// TIA Portal V20 export
// export: Created 2025-12-01T14:57:38.3565208Z, ExportSetting None, DisplayName Totally Integrated Automation Portal, DisplayVersion V20 Update 3, DisplayName TIA Portal Openness, DisplayVersion V20 Update 3, DisplayName TIA Portal Version Control Interface, DisplayVersion V20 Update 3, DisplayName STEP 7 Professional, DisplayVersion V20 Update 3, DisplayName STEP 7 Safety, DisplayVersion V20 Update 2, DisplayName WinCC Basic/Comfort/Advanced, DisplayVersion V20 Update 3, DisplayName WinCC Professional, DisplayVersion V20 Update 3, DisplayName WinCC Unified, DisplayVersion V20 Update 3
FUNCTION_BLOCK "FB73_MesaBanda_DesPaletizadorCajasPlasticco"   // FB73, LAD
TITLE = Mesa de Banda DesPaletizador de Paletas
{ S7_Optimized_Access := 'FALSE' }
AUTHOR : DESPALET
FAMILY : FRUTA
NAME : 20161001
VERSION : 1.0
// stored: AutoNumber false, SetENOAutomatically false
   VAR_INPUT
      Mesa : UInt;   // Mesa de la FB
      Error_Tx : Bool;   // Error en el Tx
      EnTension : Bool;   // Existe Tension en la Mesa
      Termico_Tx : Bool;   // Proteccion del Tx
      pHsMx : Bool;   // pHs de la Mesa
      pHsMx_PR3 : Bool;   // pHs de Protrusion de la Mesa. Nota: No existe >> ON
      Avance_Tx : Bool;   // Avance del Tx
      Termico_MBanda : Bool;   // Proteccion de la Mesa de la Banda
      MBanda_IN : Bool;   // Pos.Dentro >>> Mesa de la Banda
      MBanda_OUT : Bool;   // Pos. Fuera >>> Mesa de la Banda
      MBanda_CORTE_IN : Bool;   // Corte Dentro >>> Mesa de la Banda
      MBanda_CORTE_OUT : Bool;   // Corte Fuera >>> Mesa de la Banda
      MBanda_EM_IN : Bool;   // Emergencia Fuera >>> Mesa de la Banda
      MBanda_EM_OUT : Bool;   // Emergencia Dentro >>> Mesa de la Banda
      MBanda_EnMovimiento : Bool;   // En Movimiento >>> Mesa de la Banda
      Aviso_DesPaletizado : Bool;   // Aviso DesPaletizado >>> Interlock Rodillos
      PTF_Mx_MSig : Bool;   // S3 >> Mesa Siguiente PTF
      FTF_Mx_MSig : Bool;   // S3 >> Mesa Siguiente FTF
      MSig_CargaAct : Bool;
      Mx_VelocidadLenta_In : Bool;   // Forzar a Velociada Lenta
      F_EnvMens_Mx : Bool;   // Fin de Envio de Mensaje
      OrdSal_S03 : Bool;   // Orden de Salida por S3
      V_CNT_pHsMx : Int := 500;   // Valor de Presencia
      V_CNT_ApHsMx : Int := 500;   // Valor de Ausencia
      V_CNTSeg_ApHsMx : Int := 2000;   // Valor de Seguriadad para Ausencia
      V_TOut_Tx_Mx : Int := 15000;   // TimeOut de Entrada por E1
      V_TOut_MBanda : Int := 10000;   // TimeOut de la Mesa de la Banda
      V_TMP_Protrusion : Int := 200;   // TMP de Protrusion
      V_CNT_PerdidapHs : Int := 1000;   // CNT de Perdida de pHs
   END_VAR
   VAR_OUTPUT
      P_EnvMens_PMx : Bool;   // Permiso de Enviar Mensaje de Presencia
      P_RecepOK_Mx : Bool;   // Recepcion OK
      Permiso_DesPaletizado : Bool;   // Permiso DesPaletizado >>> Interlock Rodillos
      AVTF_Mx_MSig : Bool;   // S3 >> Mesa Siguiente AVTF
      P_Mens_Mx_MSig : Bool;   // S3 >> Mesa Siguiente P_Mens
   END_VAR
   VAR
      Anular_prE1 : Bool;   // ???
      Anular_prS3 : Bool;   // ???
      Mx_ET00 : Bool;
      Mx_ET01 : Bool;
      Mx_ET02 : Bool;
      Mx_ET08 : Bool;
      Mx_ET09 : Bool;
      Mx_ET10 : Bool;
      Mx_ET11 : Bool;
      Mx_ET12 : Bool;
      Mx_ET13 : Bool;
      Mx_ET110 : Bool;
      Mx_ET111 : Bool;
      Mx_ET50 : Bool;
      Mx_ET51 : Bool;
      Mx_ET52 : Bool;
      Mx_ET150 : Bool;
      Mx_ET151 : Bool;
      ProtocoloIniciado : Bool;   // Iniciado el Envio del Mensaje de Presencia
      MemoriaCorte_IN : Bool;   // Memoria >>> Corte Dentro >>> Mesa de la Banda
      MemoriaCorte_OUT : Bool;   // Memoria >>> Corte Fuera >>> Mesa de la Banda
      CNT_pHsMx { S7_SetPoint := 'True'} : "FB910_CNT_UHS";   // CNT de la Presencia
      CNT_ApHsMx { S7_SetPoint := 'True'} : "FB910_CNT_UHS";   // CNT de la Ausencia
      CNTSeg_ApHsMx { S7_SetPoint := 'True'} : "FB910_CNT_UHS";   // CNT de Seguridad de la Ausencia
      TMP_EnTension { ExternalAccessible := 'False'; ExternalVisible := 'False'; ExternalWritable := 'False'; S7_SetPoint := 'True'} : "FB910_CNT_UHS";
      TOut_Av_Mx { S7_SetPoint := 'True'} : "FB910_CNT_UHS";   // Time Out de Entrada de E1
      TOut_MBanda { S7_SetPoint := 'True'} : "FB910_CNT_UHS";   // Time Out de Sacar o Recoger la Mesa de la Banda
      TMP_Protrusion { S7_SetPoint := 'True'} : "FB910_CNT_UHS";   // TMP de la Protrusion
      CNT_PerdidapHs { S7_SetPoint := 'True'} : "FB910_CNT_UHS";   // CNT de Perdida de pHs
      STAT_EnvMens_PMx : Bool;   // Interna >> Envio del Mensaje de Presencia
      STAT_AVTF_Mx_MSig : Bool;   // Interna >> AVTF de Mx >> MSig
      MA_Sacar_MBanda : Bool;   // ???
      MA_Recoger_MBanda : Bool;   // ???
      VelocidadLenta_MBanda : Bool;   // ???
   END_VAR
   VAR_TEMP
      EstadoZona : "EstadoZona";   // Estado de Zona de la Mesa
      EstadoVI : "EstadosMesa";   // Estado del Vehiculo Inteliguente de la Mesa
      EstadoMAQ : "EstadoMaquina_MesaBanda_DesPaletizadorCajasPlasticco";   // Estado del Vehiculo Inteliguente de la Maquina
      ConfigFB : "UDT_ConfigFB";   // Configuracion de la FB de la Mesa
      V_Protrusion : Int;
      Aux_ET00 : Bool;
   END_VAR
BEGIN

REGION Network 1: INICIALIZAR - Recoger las Variables de Estado de la Mesa
   // Se recoge - Estado_CBx
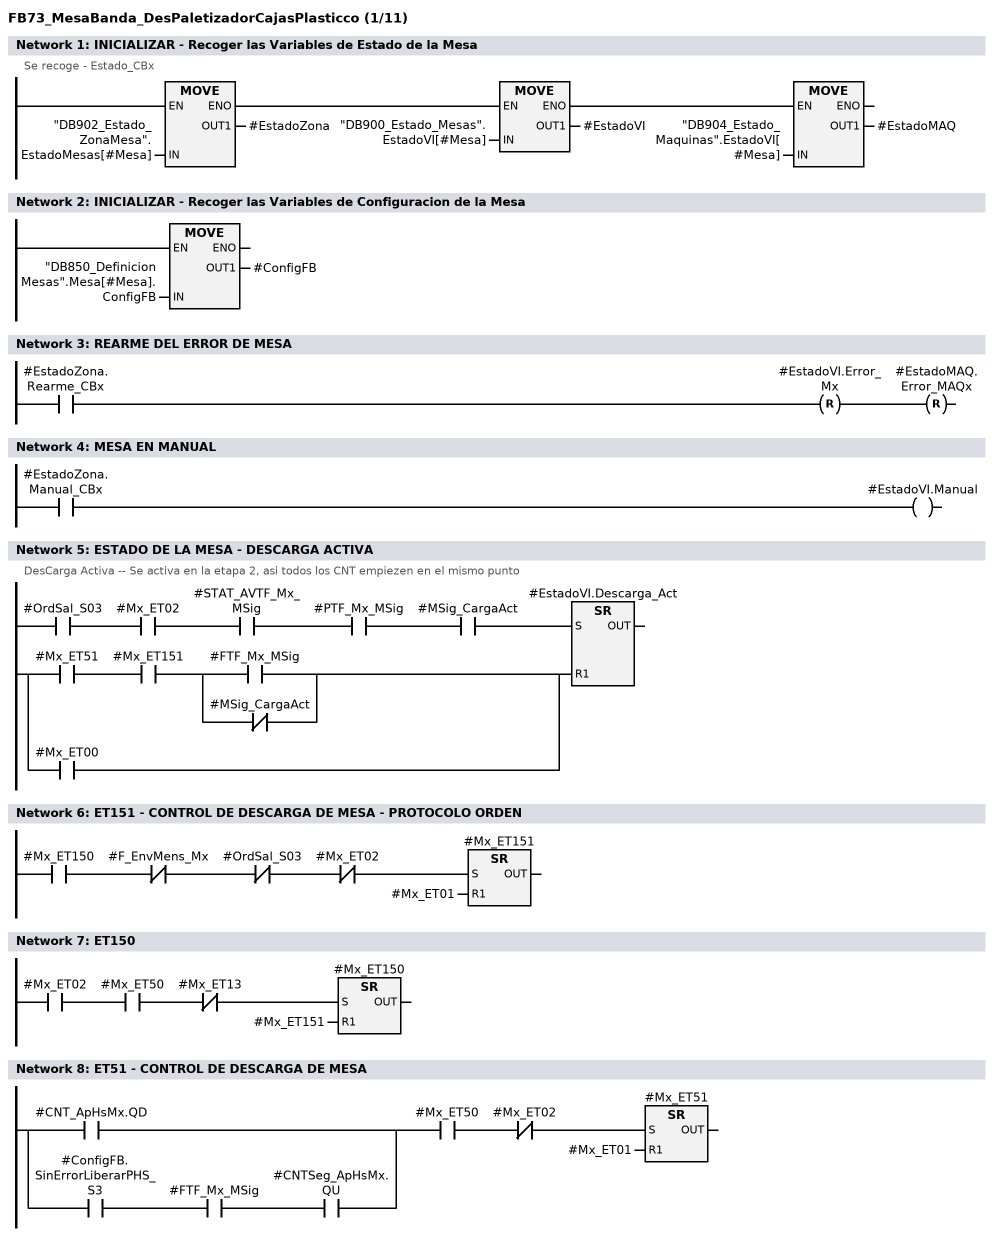
   RUNG wire#powerrail
      Move(in := "DB902_Estado_ZonaMesa".EstadoMesas[#Mesa], out1 => #EstadoZona)
      Move(in := "DB900_Estado_Mesas".EstadoVI[#Mesa], out1 => #EstadoVI)
      Move(in := "DB904_Estado_Maquinas".EstadoVI[#Mesa], out1 => #EstadoMAQ)
   END_RUNG
   // the same network as SCL:
   #EstadoZona := "DB902_Estado_ZonaMesa".EstadoMesas[#Mesa];
   #EstadoVI := "DB900_Estado_Mesas".EstadoVI[#Mesa];
   #EstadoMAQ := "DB904_Estado_Maquinas".EstadoVI[#Mesa];
END_REGION

REGION Network 2: INICIALIZAR - Recoger las Variables de Configuracion de la Mesa
   RUNG wire#powerrail
      Move(in := "DB850_DefinicionMesas".Mesa[#Mesa].ConfigFB, out1 => #ConfigFB)
   END_RUNG
   // the same network as SCL:
   #ConfigFB := "DB850_DefinicionMesas".Mesa[#Mesa].ConfigFB;
END_REGION

REGION Network 3: REARME DEL ERROR DE MESA
   RUNG wire#powerrail
      Contact( #EstadoZona.Rearme_CBx )
      R_Coil( #EstadoVI.Error_Mx )
      R_Coil( #EstadoMAQ.Error_MAQx )
   END_RUNG
   // the same network as SCL:
   IF #EstadoZona.Rearme_CBx THEN
       #EstadoVI.Error_Mx := FALSE;
       #EstadoMAQ.Error_MAQx := FALSE;
   END_IF;
END_REGION

REGION Network 4: MESA EN MANUAL
   RUNG wire#powerrail
      Contact( #EstadoZona.Manual_CBx )
      Coil( #EstadoVI.Manual )
   END_RUNG
   // the same network as SCL:
   #EstadoVI.Manual := #EstadoZona.Manual_CBx;
END_REGION

REGION Network 5: ESTADO DE LA MESA - DESCARGA ACTIVA
   // DesCarga Activa -- Se activa en la etapa 2, asi todos los CNT empiezen en el mismo punto
   RUNG wire#powerrail
      Contact( #OrdSal_S03 )
      Contact( #Mx_ET02 )
      Contact( #STAT_AVTF_Mx_MSig )
      Contact( #PTF_Mx_MSig )
      Contact( #MSig_CargaAct )
      S_SR(operand := #EstadoVI.Descarga_Act, r1 := wire#w2)
   END_RUNG
   RUNG wire#powerrail
      Contact( #Mx_ET51 )
      Contact( #Mx_ET151 )
      wire#w1
      Contact( #FTF_Mx_MSig )
   END_RUNG wire#w2
   RUNG wire#w1
      I_Contact( #MSig_CargaAct )
   END_RUNG wire#w2
   RUNG wire#powerrail
      Contact( #Mx_ET00 )
   END_RUNG wire#w2
   // the same network as SCL:
   IF #OrdSal_S03 AND #Mx_ET02 AND #STAT_AVTF_Mx_MSig AND #PTF_Mx_MSig AND #MSig_CargaAct THEN
       #EstadoVI.Descarga_Act := TRUE;   // SR flip-flop
   END_IF;
   IF (#Mx_ET51 AND #Mx_ET151 AND (#FTF_Mx_MSig OR NOT #MSig_CargaAct)) OR #Mx_ET00 THEN
       #EstadoVI.Descarga_Act := FALSE;
   END_IF;
END_REGION

REGION Network 6: ET151 - CONTROL DE DESCARGA DE MESA - PROTOCOLO ORDEN
   RUNG wire#powerrail
      Contact( #Mx_ET150 )
      I_Contact( #F_EnvMens_Mx )
      I_Contact( #OrdSal_S03 )
      I_Contact( #Mx_ET02 )
      S_SR(operand := #Mx_ET151, r1 := #Mx_ET01)
   END_RUNG
   // the same network as SCL:
   IF #Mx_ET150 AND NOT #F_EnvMens_Mx AND NOT #OrdSal_S03 AND NOT #Mx_ET02 THEN
       #Mx_ET151 := TRUE;   // SR flip-flop
   END_IF;
   IF #Mx_ET01 THEN #Mx_ET151 := FALSE; END_IF;
END_REGION

REGION Network 7: ET150
   RUNG wire#powerrail
      Contact( #Mx_ET02 )
      Contact( #Mx_ET50 )
      I_Contact( #Mx_ET13 )
      S_SR(operand := #Mx_ET150, r1 := #Mx_ET151)
   END_RUNG
   // the same network as SCL:
   IF #Mx_ET02 AND #Mx_ET50 AND NOT #Mx_ET13 THEN
       #Mx_ET150 := TRUE;   // SR flip-flop
   END_IF;
   IF #Mx_ET151 THEN #Mx_ET150 := FALSE; END_IF;
END_REGION

REGION Network 8: ET51 - CONTROL DE DESCARGA DE MESA
   RUNG wire#powerrail
      Contact( #CNT_ApHsMx.QD )
      wire#w1
      Contact( #Mx_ET50 )
      I_Contact( #Mx_ET02 )
      S_SR(operand := #Mx_ET51, r1 := #Mx_ET01)
   END_RUNG
   RUNG wire#powerrail
      Contact( #ConfigFB.SinErrorLiberarPHS_S3 )
      Contact( #FTF_Mx_MSig )
      Contact( #CNTSeg_ApHsMx.QU )
   END_RUNG wire#w1
   // the same network as SCL:
   IF (#CNT_ApHsMx.QD OR (#ConfigFB.SinErrorLiberarPHS_S3 AND #FTF_Mx_MSig AND #CNTSeg_ApHsMx.QU)) AND #Mx_ET50 AND NOT #Mx_ET02 THEN
       #Mx_ET51 := TRUE;   // SR flip-flop
   END_IF;
   IF #Mx_ET01 THEN #Mx_ET51 := FALSE; END_IF;
END_REGION

REGION Network 9: ET50
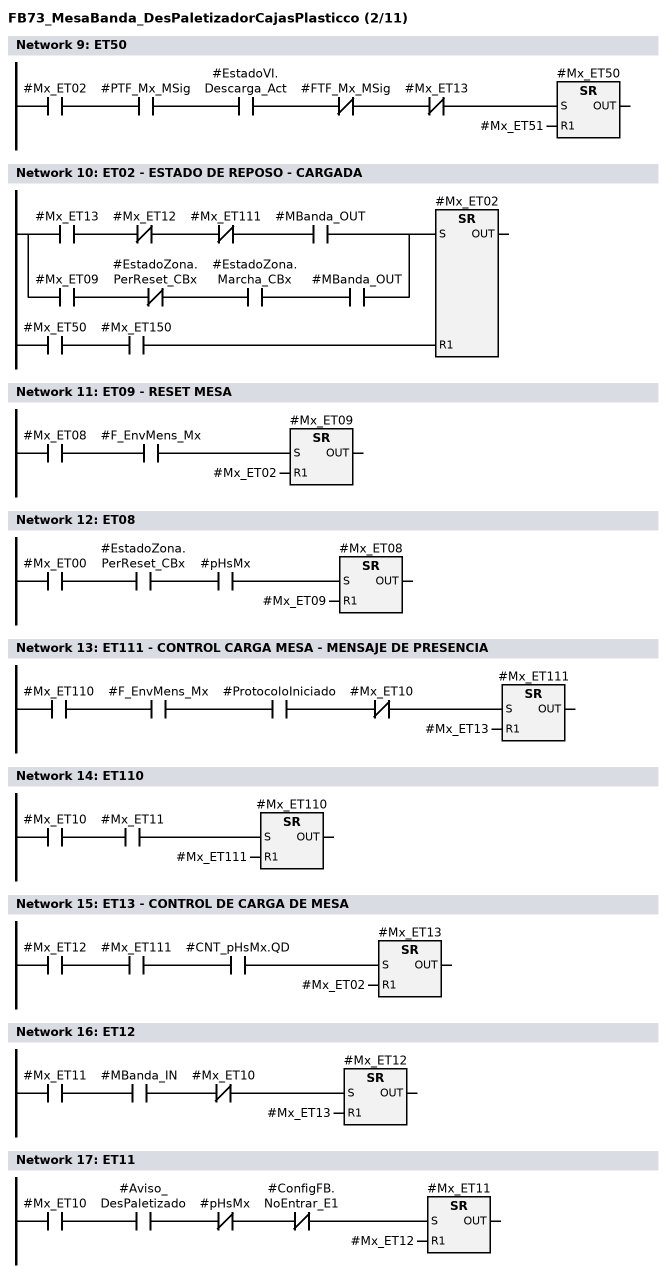
   RUNG wire#powerrail
      Contact( #Mx_ET02 )
      Contact( #PTF_Mx_MSig )
      Contact( #EstadoVI.Descarga_Act )
      I_Contact( #FTF_Mx_MSig )
      I_Contact( #Mx_ET13 )
      S_SR(operand := #Mx_ET50, r1 := #Mx_ET51)
   END_RUNG
   // the same network as SCL:
   IF #Mx_ET02 AND #PTF_Mx_MSig AND #EstadoVI.Descarga_Act AND NOT #FTF_Mx_MSig AND NOT #Mx_ET13 THEN
       #Mx_ET50 := TRUE;   // SR flip-flop
   END_IF;
   IF #Mx_ET51 THEN #Mx_ET50 := FALSE; END_IF;
END_REGION

REGION Network 10: ET02 - ESTADO DE REPOSO - CARGADA
   RUNG wire#powerrail
      Contact( #Mx_ET13 )
      I_Contact( #Mx_ET12 )
      I_Contact( #Mx_ET111 )
      Contact( #MBanda_OUT )
      wire#w1
      S_SR(operand := #Mx_ET02, r1 := wire#w2)
   END_RUNG
   RUNG wire#powerrail
      Contact( #Mx_ET09 )
      I_Contact( #EstadoZona.PerReset_CBx )
      Contact( #EstadoZona.Marcha_CBx )
      Contact( #MBanda_OUT )
   END_RUNG wire#w1
   RUNG wire#powerrail
      Contact( #Mx_ET50 )
      Contact( #Mx_ET150 )
   END_RUNG wire#w2
   // the same network as SCL:
   IF (#Mx_ET13 AND NOT #Mx_ET12 AND NOT #Mx_ET111 AND #MBanda_OUT) OR (#Mx_ET09 AND NOT #EstadoZona.PerReset_CBx AND #EstadoZona.Marcha_CBx AND #MBanda_OUT) THEN
       #Mx_ET02 := TRUE;   // SR flip-flop
   END_IF;
   IF #Mx_ET50 AND #Mx_ET150 THEN #Mx_ET02 := FALSE; END_IF;
END_REGION

REGION Network 11: ET09 - RESET MESA
   RUNG wire#powerrail
      Contact( #Mx_ET08 )
      Contact( #F_EnvMens_Mx )
      S_SR(operand := #Mx_ET09, r1 := #Mx_ET02)
   END_RUNG
   // the same network as SCL:
   IF #Mx_ET08 AND #F_EnvMens_Mx THEN
       #Mx_ET09 := TRUE;   // SR flip-flop
   END_IF;
   IF #Mx_ET02 THEN #Mx_ET09 := FALSE; END_IF;
END_REGION

REGION Network 12: ET08
   RUNG wire#powerrail
      Contact( #Mx_ET00 )
      Contact( #EstadoZona.PerReset_CBx )
      Contact( #pHsMx )
      S_SR(operand := #Mx_ET08, r1 := #Mx_ET09)
   END_RUNG
   // the same network as SCL:
   IF #Mx_ET00 AND #EstadoZona.PerReset_CBx AND #pHsMx THEN
       #Mx_ET08 := TRUE;   // SR flip-flop
   END_IF;
   IF #Mx_ET09 THEN #Mx_ET08 := FALSE; END_IF;
END_REGION

REGION Network 13: ET111 - CONTROL CARGA MESA - MENSAJE DE PRESENCIA
   RUNG wire#powerrail
      Contact( #Mx_ET110 )
      Contact( #F_EnvMens_Mx )
      Contact( #ProtocoloIniciado )
      I_Contact( #Mx_ET10 )
      S_SR(operand := #Mx_ET111, r1 := #Mx_ET13)
   END_RUNG
   // the same network as SCL:
   IF #Mx_ET110 AND #F_EnvMens_Mx AND #ProtocoloIniciado AND NOT #Mx_ET10 THEN
       #Mx_ET111 := TRUE;   // SR flip-flop
   END_IF;
   IF #Mx_ET13 THEN #Mx_ET111 := FALSE; END_IF;
END_REGION

REGION Network 14: ET110
   RUNG wire#powerrail
      Contact( #Mx_ET10 )
      Contact( #Mx_ET11 )
      S_SR(operand := #Mx_ET110, r1 := #Mx_ET111)
   END_RUNG
   // the same network as SCL:
   IF #Mx_ET10 AND #Mx_ET11 THEN
       #Mx_ET110 := TRUE;   // SR flip-flop
   END_IF;
   IF #Mx_ET111 THEN #Mx_ET110 := FALSE; END_IF;
END_REGION

REGION Network 15: ET13 - CONTROL DE CARGA DE MESA
   RUNG wire#powerrail
      Contact( #Mx_ET12 )
      Contact( #Mx_ET111 )
      Contact( #CNT_pHsMx.QD )
      S_SR(operand := #Mx_ET13, r1 := #Mx_ET02)
   END_RUNG
   // the same network as SCL:
   IF #Mx_ET12 AND #Mx_ET111 AND #CNT_pHsMx.QD THEN
       #Mx_ET13 := TRUE;   // SR flip-flop
   END_IF;
   IF #Mx_ET02 THEN #Mx_ET13 := FALSE; END_IF;
END_REGION

REGION Network 16: ET12
   RUNG wire#powerrail
      Contact( #Mx_ET11 )
      Contact( #MBanda_IN )
      I_Contact( #Mx_ET10 )
      S_SR(operand := #Mx_ET12, r1 := #Mx_ET13)
   END_RUNG
   // the same network as SCL:
   IF #Mx_ET11 AND #MBanda_IN AND NOT #Mx_ET10 THEN
       #Mx_ET12 := TRUE;   // SR flip-flop
   END_IF;
   IF #Mx_ET13 THEN #Mx_ET12 := FALSE; END_IF;
END_REGION

REGION Network 17: ET11
   RUNG wire#powerrail
      Contact( #Mx_ET10 )
      Contact( #Aviso_DesPaletizado )
      I_Contact( #pHsMx )
      I_Contact( #ConfigFB.NoEntrar_E1 )
      S_SR(operand := #Mx_ET11, r1 := #Mx_ET12)
   END_RUNG
   // the same network as SCL:
   IF #Mx_ET10 AND #Aviso_DesPaletizado AND NOT #pHsMx AND NOT #ConfigFB.NoEntrar_E1 THEN
       #Mx_ET11 := TRUE;   // SR flip-flop
   END_IF;
   IF #Mx_ET12 THEN #Mx_ET11 := FALSE; END_IF;
END_REGION

REGION Network 18: ET10
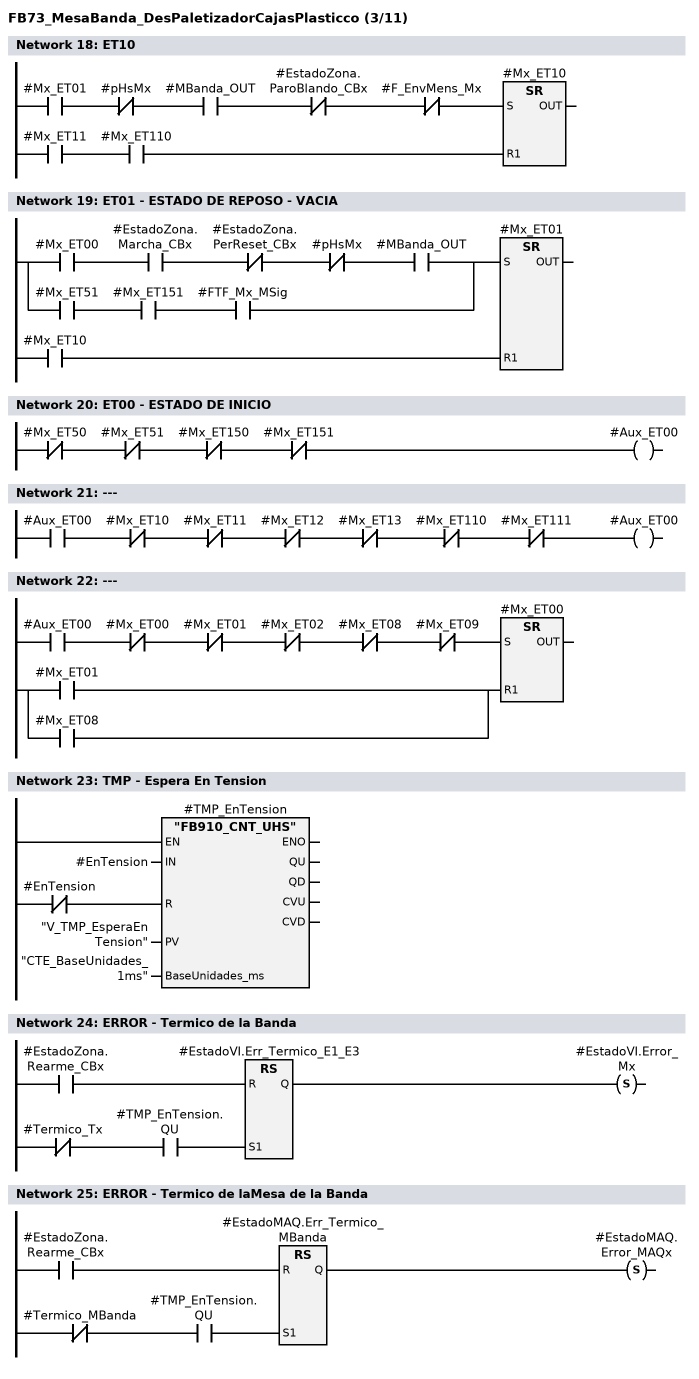
   RUNG wire#powerrail
      Contact( #Mx_ET01 )
      I_Contact( #pHsMx )
      Contact( #MBanda_OUT )
      I_Contact( #EstadoZona.ParoBlando_CBx )
      I_Contact( #F_EnvMens_Mx )
      S_SR(operand := #Mx_ET10, r1 := wire#w1)
   END_RUNG
   RUNG wire#powerrail
      Contact( #Mx_ET11 )
      Contact( #Mx_ET110 )
   END_RUNG wire#w1
   // the same network as SCL:
   IF #Mx_ET01 AND NOT #pHsMx AND #MBanda_OUT AND NOT #EstadoZona.ParoBlando_CBx AND NOT #F_EnvMens_Mx THEN
       #Mx_ET10 := TRUE;   // SR flip-flop
   END_IF;
   IF #Mx_ET11 AND #Mx_ET110 THEN #Mx_ET10 := FALSE; END_IF;
END_REGION

REGION Network 19: ET01 - ESTADO DE REPOSO - VACIA
   RUNG wire#powerrail
      Contact( #Mx_ET00 )
      Contact( #EstadoZona.Marcha_CBx )
      I_Contact( #EstadoZona.PerReset_CBx )
      I_Contact( #pHsMx )
      Contact( #MBanda_OUT )
      wire#w1
      S_SR(operand := #Mx_ET01, r1 := wire#w2)
   END_RUNG
   RUNG wire#powerrail
      Contact( #Mx_ET51 )
      Contact( #Mx_ET151 )
      Contact( #FTF_Mx_MSig )
   END_RUNG wire#w1
   RUNG wire#powerrail
      Contact( #Mx_ET10 )
   END_RUNG wire#w2
   // the same network as SCL:
   IF (#Mx_ET00 AND #EstadoZona.Marcha_CBx AND NOT #EstadoZona.PerReset_CBx AND NOT #pHsMx AND #MBanda_OUT) OR (#Mx_ET51 AND #Mx_ET151 AND #FTF_Mx_MSig) THEN
       #Mx_ET01 := TRUE;   // SR flip-flop
   END_IF;
   IF #Mx_ET10 THEN #Mx_ET01 := FALSE; END_IF;
END_REGION

REGION Network 20: ET00 - ESTADO DE INICIO
   RUNG wire#powerrail
      I_Contact( #Mx_ET50 )
      I_Contact( #Mx_ET51 )
      I_Contact( #Mx_ET150 )
      I_Contact( #Mx_ET151 )
      Coil( #Aux_ET00 )
   END_RUNG
   // the same network as SCL:
   #Aux_ET00 := NOT #Mx_ET50 AND NOT #Mx_ET51 AND NOT #Mx_ET150 AND NOT #Mx_ET151;
END_REGION

REGION Network 21: ---
   RUNG wire#powerrail
      Contact( #Aux_ET00 )
      I_Contact( #Mx_ET10 )
      I_Contact( #Mx_ET11 )
      I_Contact( #Mx_ET12 )
      I_Contact( #Mx_ET13 )
      I_Contact( #Mx_ET110 )
      I_Contact( #Mx_ET111 )
      Coil( #Aux_ET00 )
   END_RUNG
   // the same network as SCL:
   #Aux_ET00 := #Aux_ET00 AND NOT #Mx_ET10 AND NOT #Mx_ET11 AND NOT #Mx_ET12 AND NOT #Mx_ET13 AND NOT #Mx_ET110 AND NOT #Mx_ET111;
END_REGION

REGION Network 22: ---
   RUNG wire#powerrail
      Contact( #Aux_ET00 )
      I_Contact( #Mx_ET00 )
      I_Contact( #Mx_ET01 )
      I_Contact( #Mx_ET02 )
      I_Contact( #Mx_ET08 )
      I_Contact( #Mx_ET09 )
      S_SR(operand := #Mx_ET00, r1 := wire#w1)
   END_RUNG
   RUNG wire#powerrail
      Contact( #Mx_ET01 )
   END_RUNG wire#w1
   RUNG wire#powerrail
      Contact( #Mx_ET08 )
   END_RUNG wire#w1
   // the same network as SCL:
   IF #Aux_ET00 AND NOT #Mx_ET00 AND NOT #Mx_ET01 AND NOT #Mx_ET02 AND NOT #Mx_ET08 AND NOT #Mx_ET09 THEN
       #Mx_ET00 := TRUE;   // SR flip-flop
   END_IF;
   IF #Mx_ET01 OR #Mx_ET08 THEN #Mx_ET00 := FALSE; END_IF;
END_REGION

REGION Network 23: TMP - Espera En Tension
   RUNG wire#powerrail
      #TMP_EnTension(R := wire#w1, IN := #EnTension, PV := "V_TMP_EsperaEnTension", BaseUnidades_ms := "CTE_BaseUnidades_1ms", QU =>, QD =>, CVU =>, CVD =>)
   END_RUNG
   RUNG wire#powerrail
      I_Contact( #EnTension )
   END_RUNG wire#w1
   // the same network as SCL:
   #TMP_EnTension(IN := #EnTension,   // "FB910_CNT_UHS"
                  R := NOT #EnTension,
                  PV := "V_TMP_EsperaEnTension",
                  BaseUnidades_ms := "CTE_BaseUnidades_1ms");
END_REGION

REGION Network 24: ERROR - Termico de la Banda
   RUNG wire#powerrail
      Contact( #EstadoZona.Rearme_CBx )
      S_RS(operand := #EstadoVI.Err_Termico_E1_E3, s1 := wire#w1)
      S_Coil( #EstadoVI.Error_Mx )
   END_RUNG
   RUNG wire#powerrail
      I_Contact( #Termico_Tx )
      Contact( #TMP_EnTension.QU )
   END_RUNG wire#w1
   // the same network as SCL:
   IF #EstadoZona.Rearme_CBx THEN
       #EstadoVI.Err_Termico_E1_E3 := FALSE;   // RS flip-flop
   END_IF;
   IF NOT #Termico_Tx AND #TMP_EnTension.QU THEN #EstadoVI.Err_Termico_E1_E3 := TRUE; END_IF;
   IF #EstadoVI.Err_Termico_E1_E3 THEN #EstadoVI.Error_Mx := TRUE; END_IF;
END_REGION

REGION Network 25: ERROR - Termico de laMesa de la Banda
   RUNG wire#powerrail
      Contact( #EstadoZona.Rearme_CBx )
      S_RS(operand := #EstadoMAQ.Err_Termico_MBanda, s1 := wire#w1)
      S_Coil( #EstadoMAQ.Error_MAQx )
   END_RUNG
   RUNG wire#powerrail
      I_Contact( #Termico_MBanda )
      Contact( #TMP_EnTension.QU )
   END_RUNG wire#w1
   // the same network as SCL:
   IF #EstadoZona.Rearme_CBx THEN
       #EstadoMAQ.Err_Termico_MBanda := FALSE;   // RS flip-flop
   END_IF;
   IF NOT #Termico_MBanda AND #TMP_EnTension.QU THEN #EstadoMAQ.Err_Termico_MBanda := TRUE; END_IF;
   IF #EstadoMAQ.Err_Termico_MBanda THEN #EstadoMAQ.Error_MAQx := TRUE; END_IF;
END_REGION

REGION Network 26: ERROR - Mesa Ocupada
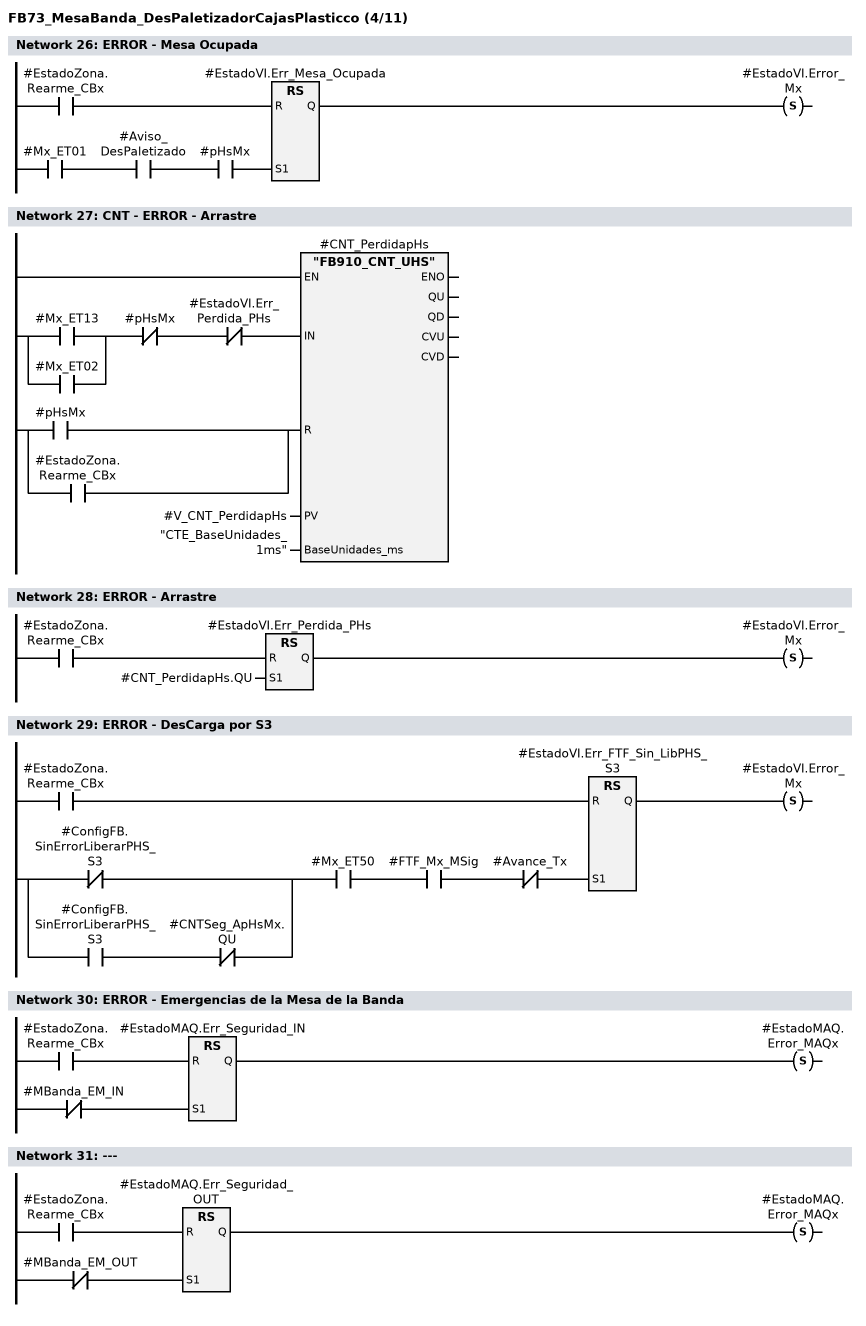
   RUNG wire#powerrail
      Contact( #EstadoZona.Rearme_CBx )
      S_RS(operand := #EstadoVI.Err_Mesa_Ocupada, s1 := wire#w1)
      S_Coil( #EstadoVI.Error_Mx )
   END_RUNG
   RUNG wire#powerrail
      Contact( #Mx_ET01 )
      Contact( #Aviso_DesPaletizado )
      Contact( #pHsMx )
   END_RUNG wire#w1
   // the same network as SCL:
   IF #EstadoZona.Rearme_CBx THEN
       #EstadoVI.Err_Mesa_Ocupada := FALSE;   // RS flip-flop
   END_IF;
   IF #Mx_ET01 AND #Aviso_DesPaletizado AND #pHsMx THEN #EstadoVI.Err_Mesa_Ocupada := TRUE; END_IF;
   IF #EstadoVI.Err_Mesa_Ocupada THEN #EstadoVI.Error_Mx := TRUE; END_IF;
END_REGION

REGION Network 27: CNT - ERROR - Arrastre
   RUNG wire#powerrail
      #CNT_PerdidapHs(IN := wire#w2, R := wire#w3, PV := #V_CNT_PerdidapHs, BaseUnidades_ms := "CTE_BaseUnidades_1ms", QU =>, QD =>, CVU =>, CVD =>)
   END_RUNG
   RUNG wire#powerrail
      Contact( #Mx_ET13 )
      wire#w1
      I_Contact( #pHsMx )
      I_Contact( #EstadoVI.Err_Perdida_PHs )
   END_RUNG wire#w2
   RUNG wire#powerrail
      Contact( #Mx_ET02 )
   END_RUNG wire#w1
   RUNG wire#powerrail
      Contact( #pHsMx )
   END_RUNG wire#w3
   RUNG wire#powerrail
      Contact( #EstadoZona.Rearme_CBx )
   END_RUNG wire#w3
   // the same network as SCL:
   #CNT_PerdidapHs(IN := (#Mx_ET13 OR #Mx_ET02) AND NOT #pHsMx AND NOT #EstadoVI.Err_Perdida_PHs,   // "FB910_CNT_UHS"
                   R := #pHsMx OR #EstadoZona.Rearme_CBx,
                   PV := #V_CNT_PerdidapHs,
                   BaseUnidades_ms := "CTE_BaseUnidades_1ms");
END_REGION

REGION Network 28: ERROR - Arrastre
   RUNG wire#powerrail
      Contact( #EstadoZona.Rearme_CBx )
      S_RS(operand := #EstadoVI.Err_Perdida_PHs, s1 := #CNT_PerdidapHs.QU)
      S_Coil( #EstadoVI.Error_Mx )
   END_RUNG
   // the same network as SCL:
   IF #EstadoZona.Rearme_CBx THEN
       #EstadoVI.Err_Perdida_PHs := FALSE;   // RS flip-flop
   END_IF;
   IF #CNT_PerdidapHs.QU THEN #EstadoVI.Err_Perdida_PHs := TRUE; END_IF;
   IF #EstadoVI.Err_Perdida_PHs THEN #EstadoVI.Error_Mx := TRUE; END_IF;
END_REGION

REGION Network 29: ERROR - DesCarga por S3
   RUNG wire#powerrail
      Contact( #EstadoZona.Rearme_CBx )
      S_RS(operand := #EstadoVI.Err_FTF_Sin_LibPHS_S3, s1 := wire#w2)
      S_Coil( #EstadoVI.Error_Mx )
   END_RUNG
   RUNG wire#powerrail
      I_Contact( #ConfigFB.SinErrorLiberarPHS_S3 )
      wire#w1
      Contact( #Mx_ET50 )
      Contact( #FTF_Mx_MSig )
      I_Contact( #Avance_Tx )
   END_RUNG wire#w2
   RUNG wire#powerrail
      Contact( #ConfigFB.SinErrorLiberarPHS_S3 )
      I_Contact( #CNTSeg_ApHsMx.QU )
   END_RUNG wire#w1
   // the same network as SCL:
   IF #EstadoZona.Rearme_CBx THEN
       #EstadoVI.Err_FTF_Sin_LibPHS_S3 := FALSE;   // RS flip-flop
   END_IF;
   IF (NOT #ConfigFB.SinErrorLiberarPHS_S3 OR (#ConfigFB.SinErrorLiberarPHS_S3 AND NOT #CNTSeg_ApHsMx.QU)) AND #Mx_ET50 AND #FTF_Mx_MSig AND NOT #Avance_Tx THEN
       #EstadoVI.Err_FTF_Sin_LibPHS_S3 := TRUE;
   END_IF;
   IF #EstadoVI.Err_FTF_Sin_LibPHS_S3 THEN #EstadoVI.Error_Mx := TRUE; END_IF;
END_REGION

REGION Network 30: ERROR - Emergencias de la Mesa de la Banda
   RUNG wire#powerrail
      Contact( #EstadoZona.Rearme_CBx )
      S_RS(operand := #EstadoMAQ.Err_Seguridad_IN, s1 := wire#w1)
      S_Coil( #EstadoMAQ.Error_MAQx )
   END_RUNG
   RUNG wire#powerrail
      I_Contact( #MBanda_EM_IN )
   END_RUNG wire#w1
   // the same network as SCL:
   IF #EstadoZona.Rearme_CBx THEN
       #EstadoMAQ.Err_Seguridad_IN := FALSE;   // RS flip-flop
   END_IF;
   IF NOT #MBanda_EM_IN THEN #EstadoMAQ.Err_Seguridad_IN := TRUE; END_IF;
   IF #EstadoMAQ.Err_Seguridad_IN THEN #EstadoMAQ.Error_MAQx := TRUE; END_IF;
END_REGION

REGION Network 31: ---
   RUNG wire#powerrail
      Contact( #EstadoZona.Rearme_CBx )
      S_RS(operand := #EstadoMAQ.Err_Seguridad_OUT, s1 := wire#w1)
      S_Coil( #EstadoMAQ.Error_MAQx )
   END_RUNG
   RUNG wire#powerrail
      I_Contact( #MBanda_EM_OUT )
   END_RUNG wire#w1
   // the same network as SCL:
   IF #EstadoZona.Rearme_CBx THEN
       #EstadoMAQ.Err_Seguridad_OUT := FALSE;   // RS flip-flop
   END_IF;
   IF NOT #MBanda_EM_OUT THEN #EstadoMAQ.Err_Seguridad_OUT := TRUE; END_IF;
   IF #EstadoMAQ.Err_Seguridad_OUT THEN #EstadoMAQ.Error_MAQx := TRUE; END_IF;
END_REGION

REGION Network 32: TMP - ERROR - TimeOut Avance
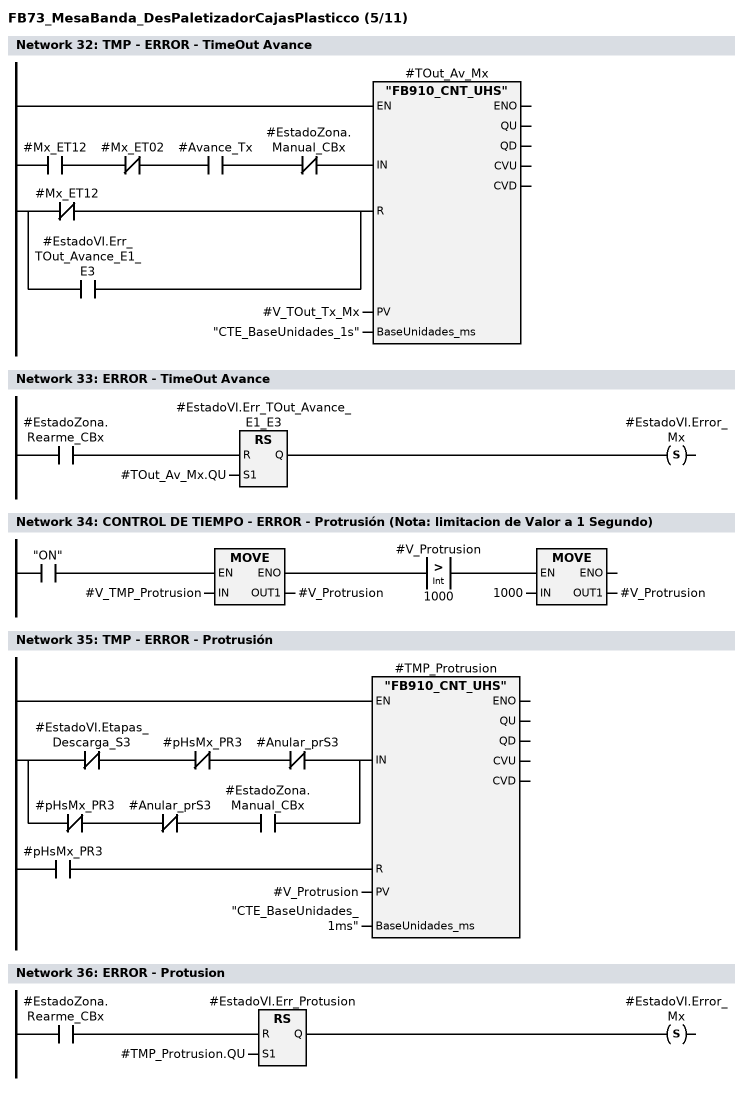
   RUNG wire#powerrail
      #TOut_Av_Mx(IN := wire#w1, R := wire#w2, PV := #V_TOut_Tx_Mx, BaseUnidades_ms := "CTE_BaseUnidades_1s", QU =>, QD =>, CVU =>, CVD =>)
   END_RUNG
   RUNG wire#powerrail
      Contact( #Mx_ET12 )
      I_Contact( #Mx_ET02 )
      Contact( #Avance_Tx )
      I_Contact( #EstadoZona.Manual_CBx )
   END_RUNG wire#w1
   RUNG wire#powerrail
      I_Contact( #Mx_ET12 )
   END_RUNG wire#w2
   RUNG wire#powerrail
      Contact( #EstadoVI.Err_TOut_Avance_E1_E3 )
   END_RUNG wire#w2
   // the same network as SCL:
   #TOut_Av_Mx(IN := #Mx_ET12 AND NOT #Mx_ET02 AND #Avance_Tx AND NOT #EstadoZona.Manual_CBx,   // "FB910_CNT_UHS"
               R := NOT #Mx_ET12 OR #EstadoVI.Err_TOut_Avance_E1_E3,
               PV := #V_TOut_Tx_Mx,
               BaseUnidades_ms := "CTE_BaseUnidades_1s");
END_REGION

REGION Network 33: ERROR - TimeOut Avance
   RUNG wire#powerrail
      Contact( #EstadoZona.Rearme_CBx )
      S_RS(operand := #EstadoVI.Err_TOut_Avance_E1_E3, s1 := #TOut_Av_Mx.QU)
      S_Coil( #EstadoVI.Error_Mx )
   END_RUNG
   // the same network as SCL:
   IF #EstadoZona.Rearme_CBx THEN
       #EstadoVI.Err_TOut_Avance_E1_E3 := FALSE;   // RS flip-flop
   END_IF;
   IF #TOut_Av_Mx.QU THEN #EstadoVI.Err_TOut_Avance_E1_E3 := TRUE; END_IF;
   IF #EstadoVI.Err_TOut_Avance_E1_E3 THEN #EstadoVI.Error_Mx := TRUE; END_IF;
END_REGION

REGION Network 34: CONTROL DE TIEMPO - ERROR - Protrusión (Nota: limitacion de Valor a 1 Segundo)
   RUNG wire#powerrail
      Contact( "ON" )
      Move(in := #V_TMP_Protrusion, out1 => #V_Protrusion)
      { S7_Templates := "SrcType := Int" } GT_Contact(in1 := #V_Protrusion, in2 := 1000)
      Move(in := 1000, out1 => #V_Protrusion)
   END_RUNG
   // the same network as SCL:
   IF "ON" THEN #V_Protrusion := #V_TMP_Protrusion; END_IF;
   IF "ON" AND (#V_Protrusion > 1000) THEN #V_Protrusion := 1000; END_IF;
END_REGION

REGION Network 35: TMP - ERROR - Protrusión
   RUNG wire#powerrail
      #TMP_Protrusion(IN := wire#w1, R := wire#w2, PV := #V_Protrusion, BaseUnidades_ms := "CTE_BaseUnidades_1ms", QU =>, QD =>, CVU =>, CVD =>)
   END_RUNG
   RUNG wire#powerrail
      I_Contact( #EstadoVI.Etapas_Descarga_S3 )
      I_Contact( #pHsMx_PR3 )
      I_Contact( #Anular_prS3 )
   END_RUNG wire#w1
   RUNG wire#powerrail
      I_Contact( #pHsMx_PR3 )
      I_Contact( #Anular_prS3 )
      Contact( #EstadoZona.Manual_CBx )
   END_RUNG wire#w1
   RUNG wire#powerrail
      Contact( #pHsMx_PR3 )
   END_RUNG wire#w2
   // the same network as SCL:
   #TMP_Protrusion(IN := (NOT #EstadoVI.Etapas_Descarga_S3 AND NOT #pHsMx_PR3 AND NOT #Anular_prS3) OR (NOT #pHsMx_PR3 AND NOT #Anular_prS3 AND #EstadoZona.Manual_CBx),   // "FB910_CNT_UHS"
                   R := #pHsMx_PR3,
                   PV := #V_Protrusion,
                   BaseUnidades_ms := "CTE_BaseUnidades_1ms");
END_REGION

REGION Network 36: ERROR - Protusion
   RUNG wire#powerrail
      Contact( #EstadoZona.Rearme_CBx )
      S_RS(operand := #EstadoVI.Err_Protusion, s1 := #TMP_Protrusion.QU)
      S_Coil( #EstadoVI.Error_Mx )
   END_RUNG
   // the same network as SCL:
   IF #EstadoZona.Rearme_CBx THEN
       #EstadoVI.Err_Protusion := FALSE;   // RS flip-flop
   END_IF;
   IF #TMP_Protrusion.QU THEN #EstadoVI.Err_Protusion := TRUE; END_IF;
   IF #EstadoVI.Err_Protusion THEN #EstadoVI.Error_Mx := TRUE; END_IF;
END_REGION

REGION Network 37: TMP - ERROR - TimeOut Recoger o Sacar la Mesa de la Banda
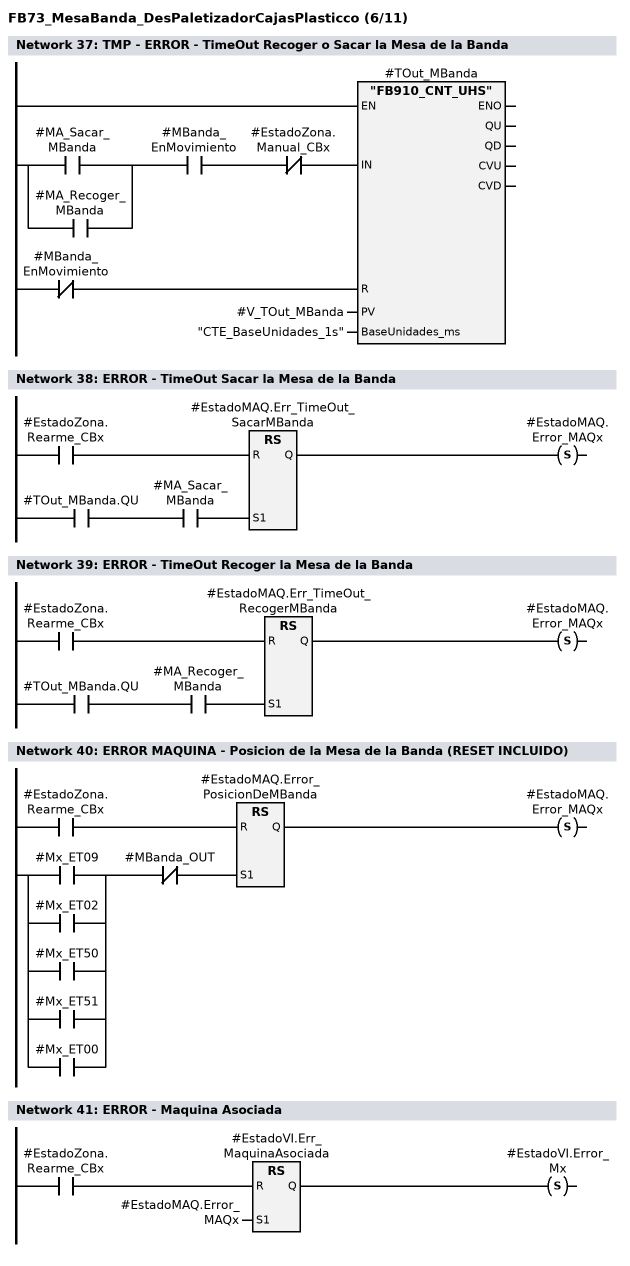
   RUNG wire#powerrail
      #TOut_MBanda(IN := wire#w2, R := wire#w3, PV := #V_TOut_MBanda, BaseUnidades_ms := "CTE_BaseUnidades_1s", QU =>, QD =>, CVU =>, CVD =>)
   END_RUNG
   RUNG wire#powerrail
      Contact( #MA_Sacar_MBanda )
      wire#w1
      Contact( #MBanda_EnMovimiento )
      I_Contact( #EstadoZona.Manual_CBx )
   END_RUNG wire#w2
   RUNG wire#powerrail
      Contact( #MA_Recoger_MBanda )
   END_RUNG wire#w1
   RUNG wire#powerrail
      I_Contact( #MBanda_EnMovimiento )
   END_RUNG wire#w3
   // the same network as SCL:
   #TOut_MBanda(IN := (#MA_Sacar_MBanda OR #MA_Recoger_MBanda) AND #MBanda_EnMovimiento AND NOT #EstadoZona.Manual_CBx,   // "FB910_CNT_UHS"
                R := NOT #MBanda_EnMovimiento,
                PV := #V_TOut_MBanda,
                BaseUnidades_ms := "CTE_BaseUnidades_1s");
END_REGION

REGION Network 38: ERROR - TimeOut Sacar la Mesa de la Banda
   RUNG wire#powerrail
      Contact( #EstadoZona.Rearme_CBx )
      S_RS(operand := #EstadoMAQ.Err_TimeOut_SacarMBanda, s1 := wire#w1)
      S_Coil( #EstadoMAQ.Error_MAQx )
   END_RUNG
   RUNG wire#powerrail
      Contact( #TOut_MBanda.QU )
      Contact( #MA_Sacar_MBanda )
   END_RUNG wire#w1
   // the same network as SCL:
   IF #EstadoZona.Rearme_CBx THEN
       #EstadoMAQ.Err_TimeOut_SacarMBanda := FALSE;   // RS flip-flop
   END_IF;
   IF #TOut_MBanda.QU AND #MA_Sacar_MBanda THEN #EstadoMAQ.Err_TimeOut_SacarMBanda := TRUE; END_IF;
   IF #EstadoMAQ.Err_TimeOut_SacarMBanda THEN #EstadoMAQ.Error_MAQx := TRUE; END_IF;
END_REGION

REGION Network 39: ERROR - TimeOut Recoger la Mesa de la Banda
   RUNG wire#powerrail
      Contact( #EstadoZona.Rearme_CBx )
      S_RS(operand := #EstadoMAQ.Err_TimeOut_RecogerMBanda, s1 := wire#w1)
      S_Coil( #EstadoMAQ.Error_MAQx )
   END_RUNG
   RUNG wire#powerrail
      Contact( #TOut_MBanda.QU )
      Contact( #MA_Recoger_MBanda )
   END_RUNG wire#w1
   // the same network as SCL:
   IF #EstadoZona.Rearme_CBx THEN
       #EstadoMAQ.Err_TimeOut_RecogerMBanda := FALSE;   // RS flip-flop
   END_IF;
   IF #TOut_MBanda.QU AND #MA_Recoger_MBanda THEN #EstadoMAQ.Err_TimeOut_RecogerMBanda := TRUE; END_IF;
   IF #EstadoMAQ.Err_TimeOut_RecogerMBanda THEN #EstadoMAQ.Error_MAQx := TRUE; END_IF;
END_REGION

REGION Network 40: ERROR MAQUINA - Posicion de la Mesa de la Banda (RESET INCLUIDO)
   RUNG wire#powerrail
      Contact( #EstadoZona.Rearme_CBx )
      S_RS(operand := #EstadoMAQ.Error_PosicionDeMBanda, s1 := wire#w2)
      S_Coil( #EstadoMAQ.Error_MAQx )
   END_RUNG
   RUNG wire#powerrail
      Contact( #Mx_ET09 )
      wire#w1
      I_Contact( #MBanda_OUT )
   END_RUNG wire#w2
   RUNG wire#powerrail
      Contact( #Mx_ET02 )
   END_RUNG wire#w1
   RUNG wire#powerrail
      Contact( #Mx_ET50 )
   END_RUNG wire#w1
   RUNG wire#powerrail
      Contact( #Mx_ET51 )
   END_RUNG wire#w1
   RUNG wire#powerrail
      Contact( #Mx_ET00 )
   END_RUNG wire#w1
   // the same network as SCL:
   IF #EstadoZona.Rearme_CBx THEN
       #EstadoMAQ.Error_PosicionDeMBanda := FALSE;   // RS flip-flop
   END_IF;
   IF (#Mx_ET09 OR #Mx_ET02 OR #Mx_ET50 OR #Mx_ET51 OR #Mx_ET00) AND NOT #MBanda_OUT THEN
       #EstadoMAQ.Error_PosicionDeMBanda := TRUE;
   END_IF;
   IF #EstadoMAQ.Error_PosicionDeMBanda THEN #EstadoMAQ.Error_MAQx := TRUE; END_IF;
END_REGION

REGION Network 41: ERROR - Maquina Asociada
   RUNG wire#powerrail
      Contact( #EstadoZona.Rearme_CBx )
      S_RS(operand := #EstadoVI.Err_MaquinaAsociada, s1 := #EstadoMAQ.Error_MAQx)
      S_Coil( #EstadoVI.Error_Mx )
   END_RUNG
   // the same network as SCL:
   IF #EstadoZona.Rearme_CBx THEN
       #EstadoVI.Err_MaquinaAsociada := FALSE;   // RS flip-flop
   END_IF;
   IF #EstadoMAQ.Error_MAQx THEN #EstadoVI.Err_MaquinaAsociada := TRUE; END_IF;
   IF #EstadoVI.Err_MaquinaAsociada THEN #EstadoVI.Error_Mx := TRUE; END_IF;
END_REGION

REGION Network 42: CONTADOR DE PRESENCIA - CNT_pHsMx
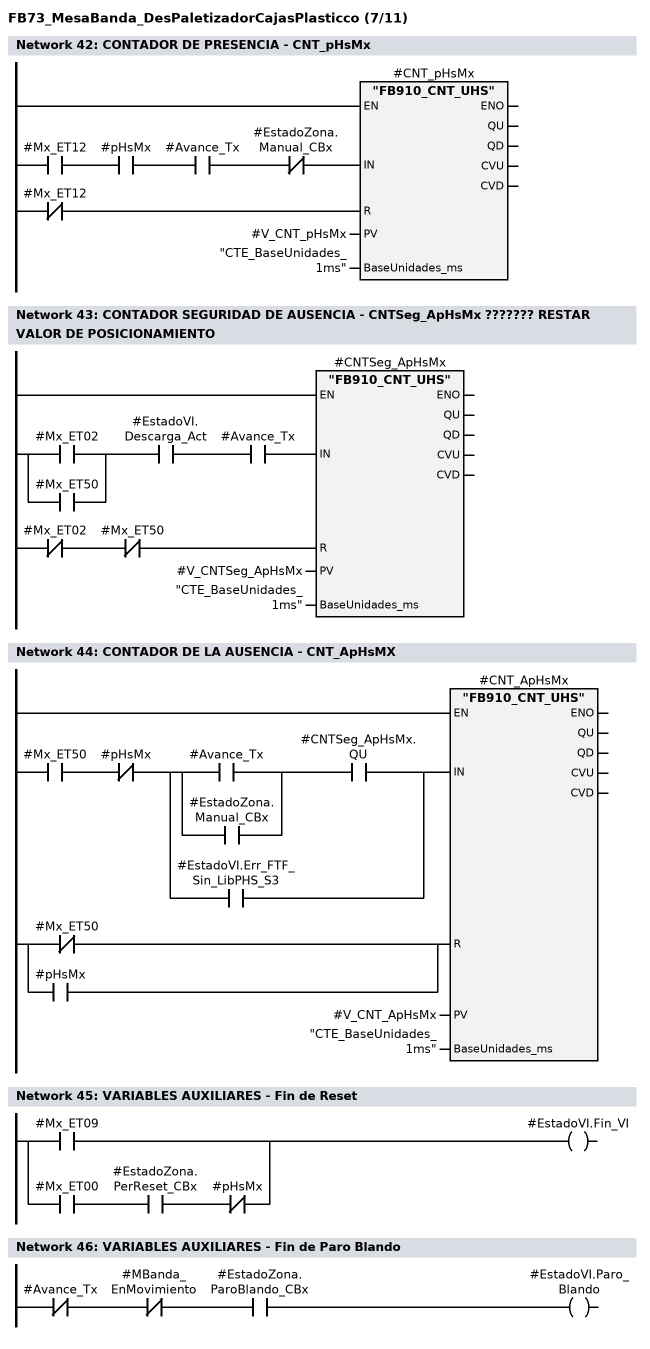
   RUNG wire#powerrail
      #CNT_pHsMx(IN := wire#w1, R := wire#w2, PV := #V_CNT_pHsMx, BaseUnidades_ms := "CTE_BaseUnidades_1ms", QU =>, QD =>, CVU =>, CVD =>)
   END_RUNG
   RUNG wire#powerrail
      Contact( #Mx_ET12 )
      Contact( #pHsMx )
      Contact( #Avance_Tx )
      I_Contact( #EstadoZona.Manual_CBx )
   END_RUNG wire#w1
   RUNG wire#powerrail
      I_Contact( #Mx_ET12 )
   END_RUNG wire#w2
   // the same network as SCL:
   #CNT_pHsMx(IN := #Mx_ET12 AND #pHsMx AND #Avance_Tx AND NOT #EstadoZona.Manual_CBx,   // "FB910_CNT_UHS"
              R := NOT #Mx_ET12,
              PV := #V_CNT_pHsMx,
              BaseUnidades_ms := "CTE_BaseUnidades_1ms");
END_REGION

REGION Network 43: CONTADOR SEGURIDAD DE AUSENCIA - CNTSeg_ApHsMx ??????? RESTAR VALOR DE POSICIONAMIENTO
   RUNG wire#powerrail
      #CNTSeg_ApHsMx(IN := wire#w2, R := wire#w3, PV := #V_CNTSeg_ApHsMx, BaseUnidades_ms := "CTE_BaseUnidades_1ms", QU =>, QD =>, CVU =>, CVD =>)
   END_RUNG
   RUNG wire#powerrail
      Contact( #Mx_ET02 )
      wire#w1
      Contact( #EstadoVI.Descarga_Act )
      Contact( #Avance_Tx )
   END_RUNG wire#w2
   RUNG wire#powerrail
      Contact( #Mx_ET50 )
   END_RUNG wire#w1
   RUNG wire#powerrail
      I_Contact( #Mx_ET02 )
      I_Contact( #Mx_ET50 )
   END_RUNG wire#w3
   // the same network as SCL:
   #CNTSeg_ApHsMx(IN := (#Mx_ET02 OR #Mx_ET50) AND #EstadoVI.Descarga_Act AND #Avance_Tx,   // "FB910_CNT_UHS"
                  R := NOT #Mx_ET02 AND NOT #Mx_ET50,
                  PV := #V_CNTSeg_ApHsMx,
                  BaseUnidades_ms := "CTE_BaseUnidades_1ms");
END_REGION

REGION Network 44: CONTADOR DE LA AUSENCIA - CNT_ApHsMX
   RUNG wire#powerrail
      #CNT_ApHsMx(IN := wire#w3, R := wire#w4, PV := #V_CNT_ApHsMx, BaseUnidades_ms := "CTE_BaseUnidades_1ms", QU =>, QD =>, CVU =>, CVD =>)
   END_RUNG
   RUNG wire#powerrail
      Contact( #Mx_ET50 )
      I_Contact( #pHsMx )
      wire#w1
      Contact( #Avance_Tx )
      wire#w2
      Contact( #CNTSeg_ApHsMx.QU )
   END_RUNG wire#w3
   RUNG wire#w1
      Contact( #EstadoZona.Manual_CBx )
   END_RUNG wire#w2
   RUNG wire#w1
      Contact( #EstadoVI.Err_FTF_Sin_LibPHS_S3 )
   END_RUNG wire#w3
   RUNG wire#powerrail
      I_Contact( #Mx_ET50 )
   END_RUNG wire#w4
   RUNG wire#powerrail
      Contact( #pHsMx )
   END_RUNG wire#w4
   // the same network as SCL:
   #CNT_ApHsMx(IN := #Mx_ET50 AND NOT #pHsMx AND (((#Avance_Tx OR #EstadoZona.Manual_CBx) AND #CNTSeg_ApHsMx.QU) OR #EstadoVI.Err_FTF_Sin_LibPHS_S3),   // "FB910_CNT_UHS"
               R := NOT #Mx_ET50 OR #pHsMx,
               PV := #V_CNT_ApHsMx,
               BaseUnidades_ms := "CTE_BaseUnidades_1ms");
END_REGION

REGION Network 45: VARIABLES AUXILIARES - Fin de Reset
   RUNG wire#powerrail
      Contact( #Mx_ET09 )
      wire#w1
      Coil( #EstadoVI.Fin_VI )
   END_RUNG
   RUNG wire#powerrail
      Contact( #Mx_ET00 )
      Contact( #EstadoZona.PerReset_CBx )
      I_Contact( #pHsMx )
   END_RUNG wire#w1
   // the same network as SCL:
   #EstadoVI.Fin_VI := #Mx_ET09 OR (#Mx_ET00 AND #EstadoZona.PerReset_CBx AND NOT #pHsMx);
END_REGION

REGION Network 46: VARIABLES AUXILIARES - Fin de Paro Blando
   RUNG wire#powerrail
      I_Contact( #Avance_Tx )
      I_Contact( #MBanda_EnMovimiento )
      Contact( #EstadoZona.ParoBlando_CBx )
      Coil( #EstadoVI.Paro_Blando )
   END_RUNG
   // the same network as SCL:
   #EstadoVI.Paro_Blando := NOT #Avance_Tx AND NOT #MBanda_EnMovimiento AND #EstadoZona.ParoBlando_CBx;
END_REGION

REGION Network 47: VARIABLES AUXILIARES - MEMORIA CORTE DE OUT >>> FUERA
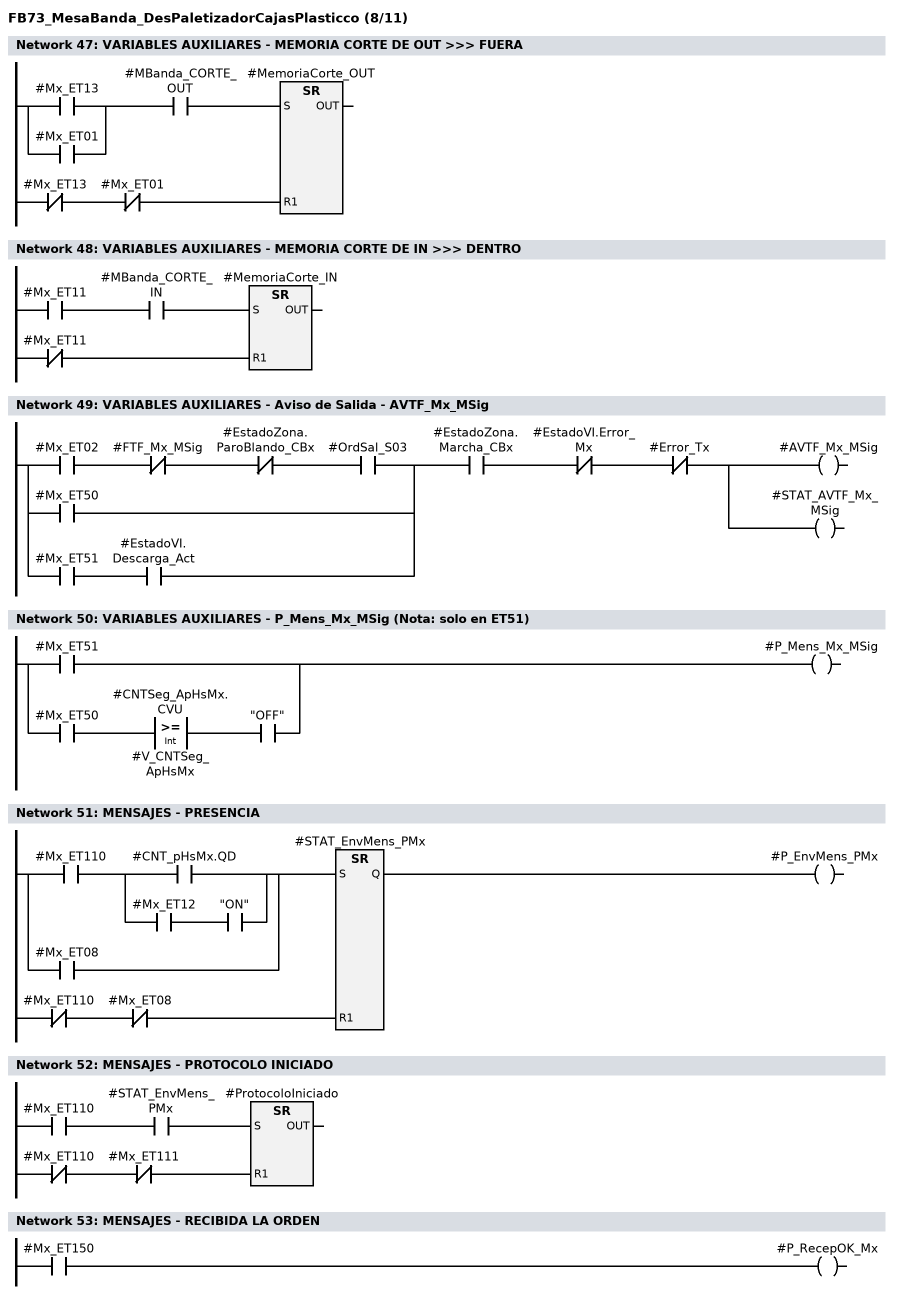
   RUNG wire#powerrail
      Contact( #Mx_ET13 )
      wire#w1
      Contact( #MBanda_CORTE_OUT )
      S_SR(operand := #MemoriaCorte_OUT, r1 := wire#w2)
   END_RUNG
   RUNG wire#powerrail
      Contact( #Mx_ET01 )
   END_RUNG wire#w1
   RUNG wire#powerrail
      I_Contact( #Mx_ET13 )
      I_Contact( #Mx_ET01 )
   END_RUNG wire#w2
   // the same network as SCL:
   IF (#Mx_ET13 OR #Mx_ET01) AND #MBanda_CORTE_OUT THEN
       #MemoriaCorte_OUT := TRUE;   // SR flip-flop
   END_IF;
   IF NOT #Mx_ET13 AND NOT #Mx_ET01 THEN #MemoriaCorte_OUT := FALSE; END_IF;
END_REGION

REGION Network 48: VARIABLES AUXILIARES - MEMORIA CORTE DE IN >>> DENTRO
   RUNG wire#powerrail
      Contact( #Mx_ET11 )
      Contact( #MBanda_CORTE_IN )
      S_SR(operand := #MemoriaCorte_IN, r1 := wire#w1)
   END_RUNG
   RUNG wire#powerrail
      I_Contact( #Mx_ET11 )
   END_RUNG wire#w1
   // the same network as SCL:
   IF #Mx_ET11 AND #MBanda_CORTE_IN THEN
       #MemoriaCorte_IN := TRUE;   // SR flip-flop
   END_IF;
   IF NOT #Mx_ET11 THEN #MemoriaCorte_IN := FALSE; END_IF;
END_REGION

REGION Network 49: VARIABLES AUXILIARES - Aviso de Salida - AVTF_Mx_MSig
   RUNG wire#powerrail
      Contact( #Mx_ET02 )
      I_Contact( #FTF_Mx_MSig )
      I_Contact( #EstadoZona.ParoBlando_CBx )
      Contact( #OrdSal_S03 )
      wire#w1
      Contact( #EstadoZona.Marcha_CBx )
      I_Contact( #EstadoVI.Error_Mx )
      I_Contact( #Error_Tx )
      wire#w2
      Coil( #AVTF_Mx_MSig )
   END_RUNG
   RUNG wire#powerrail
      Contact( #Mx_ET50 )
   END_RUNG wire#w1
   RUNG wire#powerrail
      Contact( #Mx_ET51 )
      Contact( #EstadoVI.Descarga_Act )
   END_RUNG wire#w1
   RUNG wire#w2
      Coil( #STAT_AVTF_Mx_MSig )
   END_RUNG
   // the same network as SCL:
   #AVTF_Mx_MSig := ((#Mx_ET02 AND NOT #FTF_Mx_MSig AND NOT #EstadoZona.ParoBlando_CBx AND #OrdSal_S03) OR #Mx_ET50 OR (#Mx_ET51 AND #EstadoVI.Descarga_Act)) AND #EstadoZona.Marcha_CBx AND NOT #EstadoVI.Error_Mx AND NOT #Error_Tx;
   #STAT_AVTF_Mx_MSig := #AVTF_Mx_MSig;
END_REGION

REGION Network 50: VARIABLES AUXILIARES - P_Mens_Mx_MSig (Nota: solo en ET51)
   RUNG wire#powerrail
      Contact( #Mx_ET51 )
      wire#w1
      Coil( #P_Mens_Mx_MSig )
   END_RUNG
   RUNG wire#powerrail
      Contact( #Mx_ET50 )
      { S7_Templates := "SrcType := Int" } GE_Contact(in1 := #CNTSeg_ApHsMx.CVU, in2 := #V_CNTSeg_ApHsMx)
      Contact( "OFF" )
   END_RUNG wire#w1
   // the same network as SCL:
   #P_Mens_Mx_MSig := #Mx_ET51 OR (#Mx_ET50 AND (#CNTSeg_ApHsMx.CVU >= #V_CNTSeg_ApHsMx) AND "OFF");
END_REGION

REGION Network 51: MENSAJES - PRESENCIA
   RUNG wire#powerrail
      Contact( #Mx_ET110 )
      wire#w1
      Contact( #CNT_pHsMx.QD )
      wire#w2
      S_SR(operand := #STAT_EnvMens_PMx, r1 := wire#w3)
      Coil( #P_EnvMens_PMx )
   END_RUNG
   RUNG wire#w1
      Contact( #Mx_ET12 )
      Contact( "ON" )
   END_RUNG wire#w2
   RUNG wire#powerrail
      Contact( #Mx_ET08 )
   END_RUNG wire#w2
   RUNG wire#powerrail
      I_Contact( #Mx_ET110 )
      I_Contact( #Mx_ET08 )
   END_RUNG wire#w3
   // the same network as SCL:
   IF (#Mx_ET110 AND (#CNT_pHsMx.QD OR (#Mx_ET12 AND "ON"))) OR #Mx_ET08 THEN
       #STAT_EnvMens_PMx := TRUE;   // SR flip-flop
   END_IF;
   IF NOT #Mx_ET110 AND NOT #Mx_ET08 THEN #STAT_EnvMens_PMx := FALSE; END_IF;
   #P_EnvMens_PMx := #STAT_EnvMens_PMx;
END_REGION

REGION Network 52: MENSAJES - PROTOCOLO INICIADO
   RUNG wire#powerrail
      Contact( #Mx_ET110 )
      Contact( #STAT_EnvMens_PMx )
      S_SR(operand := #ProtocoloIniciado, r1 := wire#w1)
   END_RUNG
   RUNG wire#powerrail
      I_Contact( #Mx_ET110 )
      I_Contact( #Mx_ET111 )
   END_RUNG wire#w1
   // the same network as SCL:
   IF #Mx_ET110 AND #STAT_EnvMens_PMx THEN
       #ProtocoloIniciado := TRUE;   // SR flip-flop
   END_IF;
   IF NOT #Mx_ET110 AND NOT #Mx_ET111 THEN #ProtocoloIniciado := FALSE; END_IF;
END_REGION

REGION Network 53: MENSAJES - RECIBIDA LA ORDEN
   RUNG wire#powerrail
      Contact( #Mx_ET150 )
      Coil( #P_RecepOK_Mx )
   END_RUNG
   // the same network as SCL:
   #P_RecepOK_Mx := #Mx_ET150;
END_REGION

REGION Network 54: INTERLOCK - Mesa de Rodillos del DesPaletizador de Cajas de Plastico
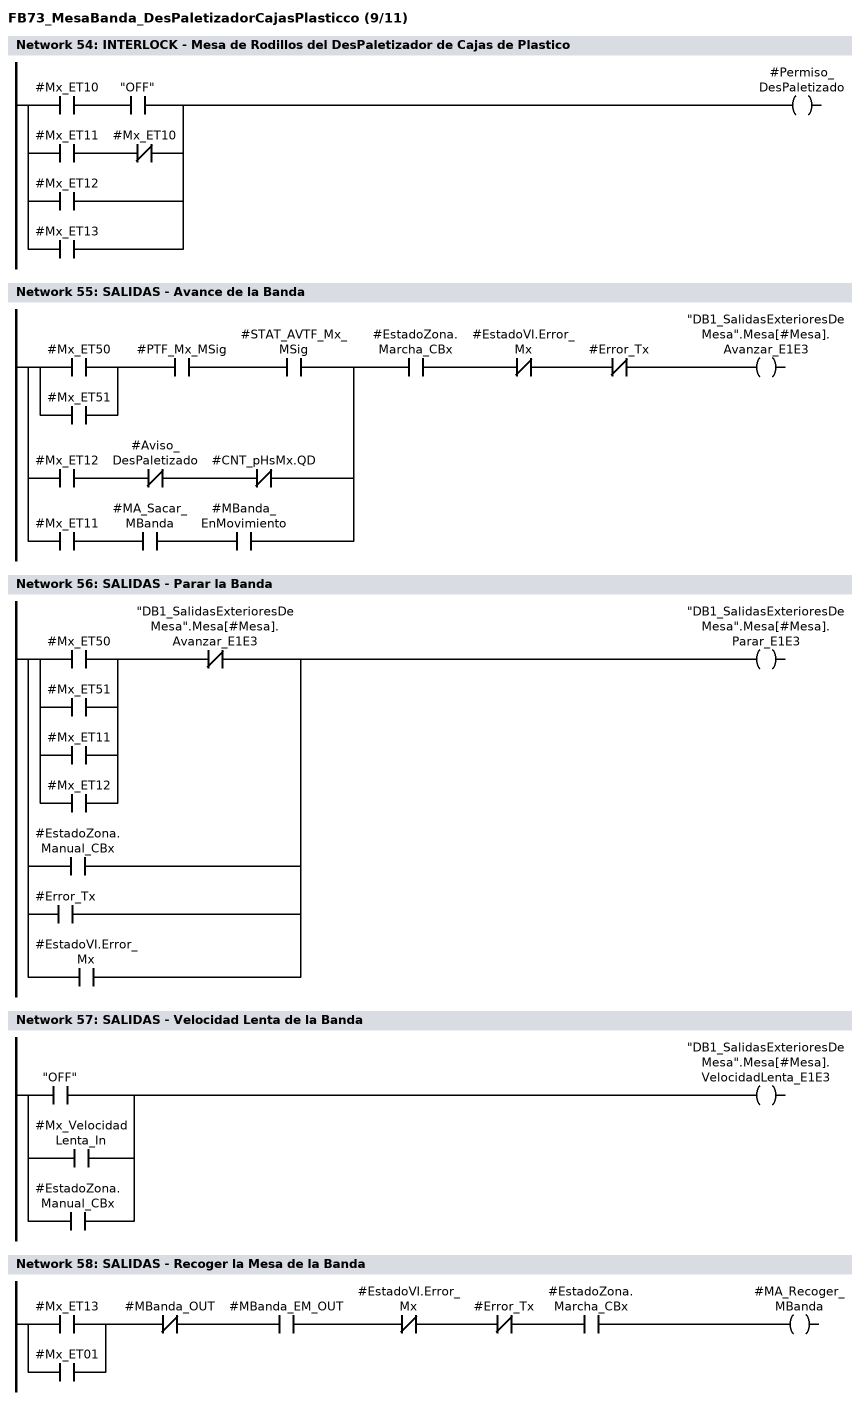
   RUNG wire#powerrail
      Contact( #Mx_ET10 )
      Contact( "OFF" )
      wire#w1
      Coil( #Permiso_DesPaletizado )
   END_RUNG
   RUNG wire#powerrail
      Contact( #Mx_ET11 )
      I_Contact( #Mx_ET10 )
   END_RUNG wire#w1
   RUNG wire#powerrail
      Contact( #Mx_ET12 )
   END_RUNG wire#w1
   RUNG wire#powerrail
      Contact( #Mx_ET13 )
   END_RUNG wire#w1
   // the same network as SCL:
   #Permiso_DesPaletizado := (#Mx_ET10 AND "OFF") OR (#Mx_ET11 AND NOT #Mx_ET10) OR #Mx_ET12 OR #Mx_ET13;
END_REGION

REGION Network 55: SALIDAS - Avance de la Banda
   RUNG wire#powerrail
      Contact( #Mx_ET50 )
      wire#w1
      Contact( #PTF_Mx_MSig )
      Contact( #STAT_AVTF_Mx_MSig )
      wire#w2
      Contact( #EstadoZona.Marcha_CBx )
      I_Contact( #EstadoVI.Error_Mx )
      I_Contact( #Error_Tx )
      Coil( "DB1_SalidasExterioresDeMesa".Mesa[#Mesa].Avanzar_E1E3 )
   END_RUNG
   RUNG wire#powerrail
      Contact( #Mx_ET51 )
   END_RUNG wire#w1
   RUNG wire#powerrail
      Contact( #Mx_ET12 )
      I_Contact( #Aviso_DesPaletizado )
      I_Contact( #CNT_pHsMx.QD )
   END_RUNG wire#w2
   RUNG wire#powerrail
      Contact( #Mx_ET11 )
      Contact( #MA_Sacar_MBanda )
      Contact( #MBanda_EnMovimiento )
   END_RUNG wire#w2
   // the same network as SCL:
   "DB1_SalidasExterioresDeMesa".Mesa[#Mesa].Avanzar_E1E3 := (((#Mx_ET50 OR #Mx_ET51) AND #PTF_Mx_MSig AND #STAT_AVTF_Mx_MSig) OR (#Mx_ET12 AND NOT #Aviso_DesPaletizado AND NOT #CNT_pHsMx.QD) OR (#Mx_ET11 AND #MA_Sacar_MBanda AND #MBanda_EnMovimiento)) AND #EstadoZona.Marcha_CBx AND NOT #EstadoVI.Error_Mx AND NOT #Error_Tx;
END_REGION

REGION Network 56: SALIDAS - Parar la Banda
   RUNG wire#powerrail
      Contact( #Mx_ET50 )
      wire#w1
      I_Contact( "DB1_SalidasExterioresDeMesa".Mesa[#Mesa].Avanzar_E1E3 )
      wire#w2
      Coil( "DB1_SalidasExterioresDeMesa".Mesa[#Mesa].Parar_E1E3 )
   END_RUNG
   RUNG wire#powerrail
      Contact( #Mx_ET51 )
   END_RUNG wire#w1
   RUNG wire#powerrail
      Contact( #Mx_ET11 )
   END_RUNG wire#w1
   RUNG wire#powerrail
      Contact( #Mx_ET12 )
   END_RUNG wire#w1
   RUNG wire#powerrail
      Contact( #EstadoZona.Manual_CBx )
   END_RUNG wire#w2
   RUNG wire#powerrail
      Contact( #Error_Tx )
   END_RUNG wire#w2
   RUNG wire#powerrail
      Contact( #EstadoVI.Error_Mx )
   END_RUNG wire#w2
   // the same network as SCL:
   "DB1_SalidasExterioresDeMesa".Mesa[#Mesa].Parar_E1E3 := ((#Mx_ET50 OR #Mx_ET51 OR #Mx_ET11 OR #Mx_ET12) AND NOT "DB1_SalidasExterioresDeMesa".Mesa[#Mesa].Avanzar_E1E3) OR #EstadoZona.Manual_CBx OR #Error_Tx OR #EstadoVI.Error_Mx;
END_REGION

REGION Network 57: SALIDAS - Velocidad Lenta de la Banda
   RUNG wire#powerrail
      Contact( "OFF" )
      wire#w1
      Coil( "DB1_SalidasExterioresDeMesa".Mesa[#Mesa].VelocidadLenta_E1E3 )
   END_RUNG
   RUNG wire#powerrail
      Contact( #Mx_VelocidadLenta_In )
   END_RUNG wire#w1
   RUNG wire#powerrail
      Contact( #EstadoZona.Manual_CBx )
   END_RUNG wire#w1
   // the same network as SCL:
   "DB1_SalidasExterioresDeMesa".Mesa[#Mesa].VelocidadLenta_E1E3 := "OFF" OR #Mx_VelocidadLenta_In OR #EstadoZona.Manual_CBx;
END_REGION

REGION Network 58: SALIDAS - Recoger la Mesa de la Banda
   RUNG wire#powerrail
      Contact( #Mx_ET13 )
      wire#w1
      I_Contact( #MBanda_OUT )
      Contact( #MBanda_EM_OUT )
      I_Contact( #EstadoVI.Error_Mx )
      I_Contact( #Error_Tx )
      Contact( #EstadoZona.Marcha_CBx )
      Coil( #MA_Recoger_MBanda )
   END_RUNG
   RUNG wire#powerrail
      Contact( #Mx_ET01 )
   END_RUNG wire#w1
   // the same network as SCL:
   #MA_Recoger_MBanda := (#Mx_ET13 OR #Mx_ET01) AND NOT #MBanda_OUT AND #MBanda_EM_OUT AND NOT #EstadoVI.Error_Mx AND NOT #Error_Tx AND #EstadoZona.Marcha_CBx;
END_REGION

REGION Network 59: SALIDAS - Sacar la Mesa de la Banda
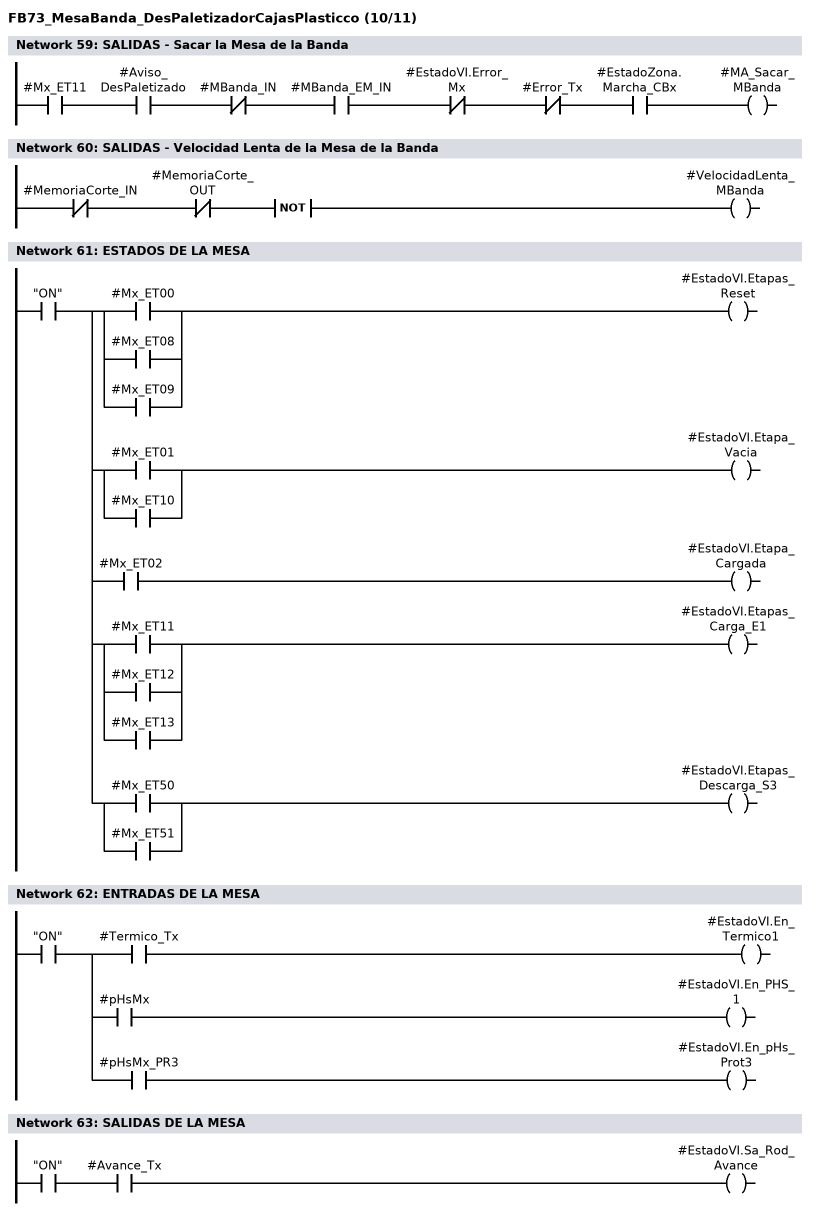
   RUNG wire#powerrail
      Contact( #Mx_ET11 )
      Contact( #Aviso_DesPaletizado )
      I_Contact( #MBanda_IN )
      Contact( #MBanda_EM_IN )
      I_Contact( #EstadoVI.Error_Mx )
      I_Contact( #Error_Tx )
      Contact( #EstadoZona.Marcha_CBx )
      Coil( #MA_Sacar_MBanda )
   END_RUNG
   // the same network as SCL:
   #MA_Sacar_MBanda := #Mx_ET11 AND #Aviso_DesPaletizado AND NOT #MBanda_IN AND #MBanda_EM_IN AND NOT #EstadoVI.Error_Mx AND NOT #Error_Tx AND #EstadoZona.Marcha_CBx;
END_REGION

REGION Network 60: SALIDAS - Velocidad Lenta de la Mesa de la Banda
   RUNG wire#powerrail
      I_Contact( #MemoriaCorte_IN )
      I_Contact( #MemoriaCorte_OUT )
      Not()
      Coil( #VelocidadLenta_MBanda )
   END_RUNG
   // the same network as SCL:
   #VelocidadLenta_MBanda := NOT (NOT #MemoriaCorte_IN AND NOT #MemoriaCorte_OUT);
END_REGION

REGION Network 61: ESTADOS DE LA MESA
   RUNG wire#powerrail
      Contact( "ON" )
      wire#w1
      Contact( #Mx_ET00 )
      wire#w2
      Coil( #EstadoVI.Etapas_Reset )
   END_RUNG
   RUNG wire#w1
      Contact( #Mx_ET08 )
   END_RUNG wire#w2
   RUNG wire#w1
      Contact( #Mx_ET09 )
   END_RUNG wire#w2
   RUNG wire#w1
      Contact( #Mx_ET01 )
      wire#w3
      Coil( #EstadoVI.Etapa_Vacia )
   END_RUNG
   RUNG wire#w1
      Contact( #Mx_ET10 )
   END_RUNG wire#w3
   RUNG wire#w1
      Contact( #Mx_ET02 )
      Coil( #EstadoVI.Etapa_Cargada )
   END_RUNG
   RUNG wire#w1
      Contact( #Mx_ET11 )
      wire#w4
      Coil( #EstadoVI.Etapas_Carga_E1 )
   END_RUNG
   RUNG wire#w1
      Contact( #Mx_ET12 )
   END_RUNG wire#w4
   RUNG wire#w1
      Contact( #Mx_ET13 )
   END_RUNG wire#w4
   RUNG wire#w1
      Contact( #Mx_ET50 )
      wire#w5
      Coil( #EstadoVI.Etapas_Descarga_S3 )
   END_RUNG
   RUNG wire#w1
      Contact( #Mx_ET51 )
   END_RUNG wire#w5
   // the same network as SCL:
   #EstadoVI.Etapas_Reset := "ON" AND (#Mx_ET00 OR #Mx_ET08 OR #Mx_ET09);
   #EstadoVI.Etapa_Vacia := "ON" AND (#Mx_ET01 OR #Mx_ET10);
   #EstadoVI.Etapa_Cargada := "ON" AND #Mx_ET02;
   #EstadoVI.Etapas_Carga_E1 := "ON" AND (#Mx_ET11 OR #Mx_ET12 OR #Mx_ET13);
   #EstadoVI.Etapas_Descarga_S3 := "ON" AND (#Mx_ET50 OR #Mx_ET51);
END_REGION

REGION Network 62: ENTRADAS DE LA MESA
   RUNG wire#powerrail
      Contact( "ON" )
      wire#w1
      Contact( #Termico_Tx )
      Coil( #EstadoVI.En_Termico1 )
   END_RUNG
   RUNG wire#w1
      Contact( #pHsMx )
      Coil( #EstadoVI.En_PHS_1 )
   END_RUNG
   RUNG wire#w1
      Contact( #pHsMx_PR3 )
      Coil( #EstadoVI.En_pHs_Prot3 )
   END_RUNG
   // the same network as SCL:
   #EstadoVI.En_Termico1 := "ON" AND #Termico_Tx;
   #EstadoVI.En_PHS_1 := "ON" AND #pHsMx;
   #EstadoVI.En_pHs_Prot3 := "ON" AND #pHsMx_PR3;
END_REGION

REGION Network 63: SALIDAS DE LA MESA
   RUNG wire#powerrail
      Contact( "ON" )
      Contact( #Avance_Tx )
      Coil( #EstadoVI.Sa_Rod_Avance )
   END_RUNG
   // the same network as SCL:
   #EstadoVI.Sa_Rod_Avance := "ON" AND #Avance_Tx;
END_REGION

REGION Network 64: ESTADOS DE LA MAQUINA (HMI)
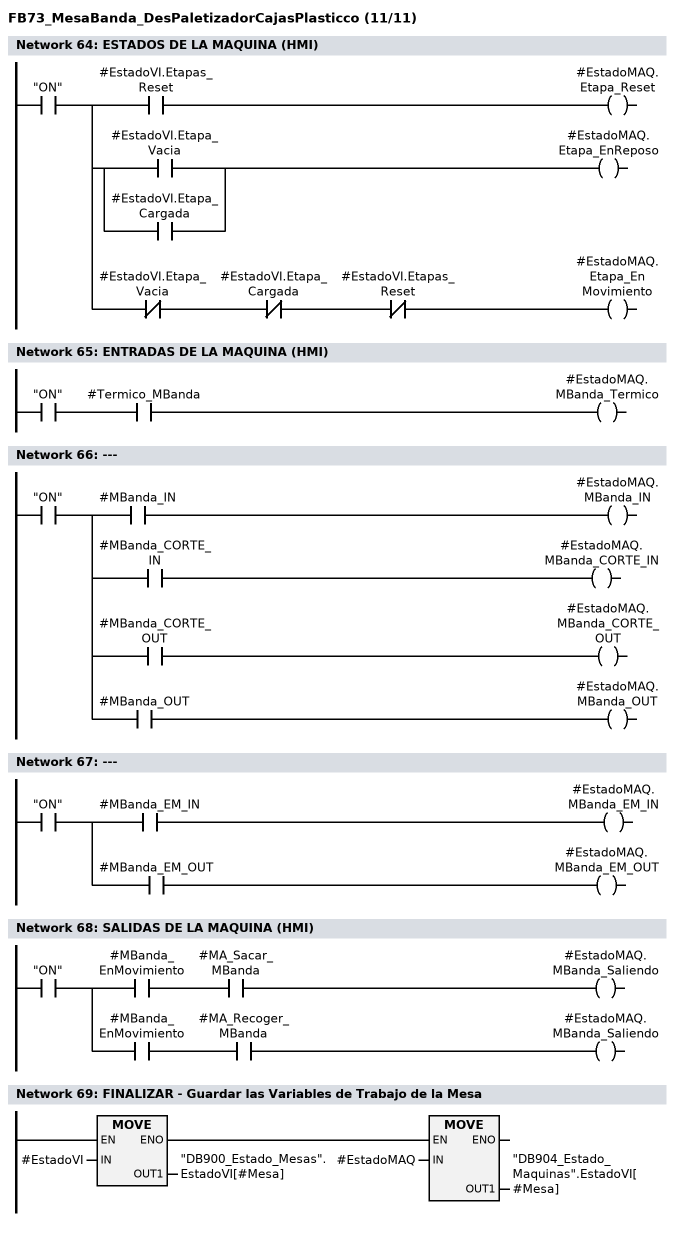
   RUNG wire#powerrail
      Contact( "ON" )
      wire#w1
      Contact( #EstadoVI.Etapas_Reset )
      Coil( #EstadoMAQ.Etapa_Reset )
   END_RUNG
   RUNG wire#w1
      Contact( #EstadoVI.Etapa_Vacia )
      wire#w2
      Coil( #EstadoMAQ.Etapa_EnReposo )
   END_RUNG
   RUNG wire#w1
      Contact( #EstadoVI.Etapa_Cargada )
   END_RUNG wire#w2
   RUNG wire#w1
      I_Contact( #EstadoVI.Etapa_Vacia )
      I_Contact( #EstadoVI.Etapa_Cargada )
      I_Contact( #EstadoVI.Etapas_Reset )
      Coil( #EstadoMAQ.Etapa_EnMovimiento )
   END_RUNG
   // the same network as SCL:
   #EstadoMAQ.Etapa_Reset := "ON" AND #EstadoVI.Etapas_Reset;
   #EstadoMAQ.Etapa_EnReposo := "ON" AND (#EstadoVI.Etapa_Vacia OR #EstadoVI.Etapa_Cargada);
   #EstadoMAQ.Etapa_EnMovimiento := "ON" AND NOT #EstadoVI.Etapa_Vacia AND NOT #EstadoVI.Etapa_Cargada AND NOT #EstadoVI.Etapas_Reset;
END_REGION

REGION Network 65: ENTRADAS DE LA MAQUINA (HMI)
   RUNG wire#powerrail
      Contact( "ON" )
      Contact( #Termico_MBanda )
      Coil( #EstadoMAQ.MBanda_Termico )
   END_RUNG
   // the same network as SCL:
   #EstadoMAQ.MBanda_Termico := "ON" AND #Termico_MBanda;
END_REGION

REGION Network 66: ---
   RUNG wire#powerrail
      Contact( "ON" )
      wire#w1
      Contact( #MBanda_IN )
      Coil( #EstadoMAQ.MBanda_IN )
   END_RUNG
   RUNG wire#w1
      Contact( #MBanda_CORTE_IN )
      Coil( #EstadoMAQ.MBanda_CORTE_IN )
   END_RUNG
   RUNG wire#w1
      Contact( #MBanda_CORTE_OUT )
      Coil( #EstadoMAQ.MBanda_CORTE_OUT )
   END_RUNG
   RUNG wire#w1
      Contact( #MBanda_OUT )
      Coil( #EstadoMAQ.MBanda_OUT )
   END_RUNG
   // the same network as SCL:
   #EstadoMAQ.MBanda_IN := "ON" AND #MBanda_IN;
   #EstadoMAQ.MBanda_CORTE_IN := "ON" AND #MBanda_CORTE_IN;
   #EstadoMAQ.MBanda_CORTE_OUT := "ON" AND #MBanda_CORTE_OUT;
   #EstadoMAQ.MBanda_OUT := "ON" AND #MBanda_OUT;
END_REGION

REGION Network 67: ---
   RUNG wire#powerrail
      Contact( "ON" )
      wire#w1
      Contact( #MBanda_EM_IN )
      Coil( #EstadoMAQ.MBanda_EM_IN )
   END_RUNG
   RUNG wire#w1
      Contact( #MBanda_EM_OUT )
      Coil( #EstadoMAQ.MBanda_EM_OUT )
   END_RUNG
   // the same network as SCL:
   #EstadoMAQ.MBanda_EM_IN := "ON" AND #MBanda_EM_IN;
   #EstadoMAQ.MBanda_EM_OUT := "ON" AND #MBanda_EM_OUT;
END_REGION

REGION Network 68: SALIDAS DE LA MAQUINA (HMI)
   RUNG wire#powerrail
      Contact( "ON" )
      wire#w1
      Contact( #MBanda_EnMovimiento )
      Contact( #MA_Sacar_MBanda )
      Coil( #EstadoMAQ.MBanda_Saliendo )
   END_RUNG
   RUNG wire#w1
      Contact( #MBanda_EnMovimiento )
      Contact( #MA_Recoger_MBanda )
      Coil( #EstadoMAQ.MBanda_Saliendo )
   END_RUNG
   // the same network as SCL:
   #EstadoMAQ.MBanda_Saliendo := "ON" AND #MBanda_EnMovimiento AND #MA_Sacar_MBanda;
   #EstadoMAQ.MBanda_Saliendo := "ON" AND #MBanda_EnMovimiento AND #MA_Recoger_MBanda;
END_REGION

REGION Network 69: FINALIZAR - Guardar las Variables de Trabajo de la Mesa
   RUNG wire#powerrail
      Move(in := #EstadoVI, out1 => "DB900_Estado_Mesas".EstadoVI[#Mesa])
      Move(in := #EstadoMAQ, out1 => "DB904_Estado_Maquinas".EstadoVI[#Mesa])
   END_RUNG
   // the same network as SCL:
   "DB900_Estado_Mesas".EstadoVI[#Mesa] := #EstadoVI;
   "DB904_Estado_Maquinas".EstadoVI[#Mesa] := #EstadoMAQ;
END_REGION
END_FUNCTION_BLOCK
